// Initialize component without injecting PermIntlk interfaces
// This tests the scenario where PermIntlk configuration is not provided
TestComponent[5].Initialize();

// Since we never injected PermIntlk configuration interfaces,
// they should be null (0) by default
// The component should handle this gracefully via __QUERYINTERFACE checks

// Call CyclicLogic multiple times - should not crash
TestComponent[5].CyclicLogic();
TestComponent[5].CyclicLogic();

// Try to execute a command - should handle missing PermIntlk gracefully
TestComponent[5].ExecuteCommand(CmdIndex := 1);

// Component should still function
AssertTrue(
    Condition := TestComponent[5].BaseStatus.Initialized,
    Message := 'Component should remain initialized with missing PermIntlk interface'
);

// The command execution should not cause the component to crash
AssertFalse(
    Condition := TestComponent[5].BaseStatus.Error,
    Message := 'Component should not be in error state when PermIntlk interface is missing'
);

TEST_FINISHED();
END_METHOD

METHOD PRIVATE TEST_Component_QueryInterface_ValidatesTypes
VAR
    DummyCommandInterface : I_Command;
    QueryResult : BOOL;
END_VAR
// Tier 0 Test: Verify proper use of __QUERYINTERFACE for type checking
TEST(__POUNAME());

// Use array index 16 for this test method
iTestComponent := TestComponent[16];
iTestCommand := TestCommandConfigured[16].Command;

// Initialize test objects
TestComponent[16].Initialize();
TestCommandConfigured[16].Initialize();

// Test that the command implements I_Command interface
QueryResult := __QUERYINTERFACE(
    TestCommandConfigured[16].Command,
    DummyCommandInterface
);

AssertTrue(
    Condition := QueryResult,
    Message := 'FB_Command should implement I_Command interface'
);

// Test the pattern used in the codebase: check both != 0 AND __QUERYINTERFACE
// This is the defensive programming pattern used throughout the component
// Here we test with an actual interface reference, not a FB instance
AssertTrue(
    Condition := (TestCommandConfigured[16].iCommandConfiguration <> 0) AND __QUERYINTERFACE(TestCommandConfigured[16].iCommandConfiguration, TestCommandConfigured[16].iCommandConfiguration),
    Message := 'Standard pattern: interface should be non-null AND correct type'
);

// Verify that a null interface check properly fails
// The pattern (interface <> 0) protects against null access
AssertFalse(
    Condition := (0 <> 0),  // This is always FALSE when interface is null
    Message := 'Null check (0 <> 0) should be FALSE'
);

// This shows why we need the null check BEFORE __QUERYINTERFACE
// We don't call __QUERYINTERFACE on null to avoid potential issues

TEST_FINISHED();
END_METHOD

METHOD PRIVATE TEST_ComponentConfiguration_BaseConfiguration_ReferenceValid
// Tier 0 Test: ComponentConfiguration.BaseConfiguration reference should be valid
TEST(__POUNAME());

// Use array index 6 for this test method
iTestComponent := TestComponent[6];

// Initialize component
TestComponent[6].Initialize();

// Verify reference chain is valid
AssertTrue(
    Condition := __ISVALIDREF(TestComponent[6].ComponentConfiguration.BaseConfiguration),
    Message := 'ComponentConfiguration.BaseConfiguration reference should be valid'
);

// Verify the reference works by accessing a field through it
// Check that we can access nested fields without error
AssertTrue(
    Condition := TestComponent[6].ComponentConfiguration.BaseConfiguration.LogTraceConfiguration.When >= 0,
    Message := 'Should be able to access fields through BaseConfiguration reference'
);

TEST_FINISHED();
END_METHOD

METHOD PRIVATE TEST_ComponentStatus_BaseStatus_ReferenceValid
// Tier 0 Test: ComponentStatus.BaseStatus reference should be valid after init
TEST(__POUNAME());

// Use array index 7 for this test method
iTestComponent := TestComponent[7];

// Initialize component
TestComponent[7].Initialize();

// Verify reference chain is valid
AssertTrue(
    Condition := __ISVALIDREF(TestComponent[7].ComponentStatus.BaseStatus),
    Message := 'ComponentStatus.BaseStatus reference should be valid'
);

// Verify the reference is working by checking a value through it
AssertEquals_BOOL(
    Expected := TestComponent[7].BaseStatus.Initialized,
    Actual := TestComponent[7].ComponentStatus.BaseStatus.Initialized,
    Message := 'ComponentStatus.BaseStatus should reference component BaseStatus'
);

// Verify InitComplete is accessible through the reference
AssertTrue(
    Condition := TestComponent[7].ComponentStatus.BaseStatus.Initialized,
    Message := 'Should be able to access InitComplete through reference chain'
);

TEST_FINISHED();
END_METHOD

METHOD PRIVATE GivenAbortInvokedDuringValidation_CommandNeverEnqueuedOrExecuted
TEST(__POUNAME());

TEST_FINISHED();
END_METHOD

METHOD PRIVATE GivenBusyCommandElapsedTimeEqualsTimeout_CommandAborted
TEST(__POUNAME());

TEST_FINISHED();
END_METHOD

METHOD PRIVATE GivenCommandBusyAndInterlockLostWithAbortOnInterlockDrop_AbortFires
TEST(__POUNAME());

TEST_FINISHED();
END_METHOD

METHOD PRIVATE GivenCommandBusyAndInterlockLostWithoutAbortOnInterlockDrop_CommandContinues
TEST(__POUNAME());

TEST_FINISHED();
END_METHOD

METHOD PRIVATE GivenCommandBusyAndInterlockStaysOk_NoAbortOccurs
TEST(__POUNAME());

TEST_FINISHED();
END_METHOD

METHOD PRIVATE GivenComponentBusyDuringValidation_ResultConflict
TEST(__POUNAME());

TEST_FINISHED();
END_METHOD

METHOD PRIVATE GivenIndeterminantCommandDequeuedButPermissiveDropsBeforeExecute_ResultForbiddenNotOk
TEST(__POUNAME());

TEST_FINISHED();
END_METHOD

METHOD PRIVATE GivenInterlockNotInitComplete_CommandValidationFailsForbidden
TEST(__POUNAME());

TEST_FINISHED();
END_METHOD

METHOD PRIVATE GivenPermIntlkAllRequiredItemsTrue_EvaluateOKReturnsTrue
VAR
	// Test conditions that will all be TRUE
	TestCondition1							: BOOL := TRUE;
	TestCondition2							: BOOL := TRUE;
	TestCondition3							: BOOL := TRUE;
END_VAR
TEST(__POUNAME());

// Use array index 250 for this test method
iTestPermIntlkConfig := TestPermIntlkConfig[250];
iTestPermIntlk := TestPermIntlk[250];

// Configure PermIntlk for "All Conditions Must Be Met" mode
TestPermIntlkConfig[250].P_PermIntlkConfiguration.Mode := E_ModePermIntlk.IfAllConditionsMet;

// Set up multiple conditions that are all TRUE
TestPermIntlkConfig[250].P_PermIntlkConfiguration.PermIntlkObj[1].Condition := TestCondition1; // TRUE
TestPermIntlkConfig[250].P_PermIntlkConfiguration.PermIntlkObj[1].Description := 'Test Condition 1 - Should be TRUE';

TestPermIntlkConfig[250].P_PermIntlkConfiguration.PermIntlkObj[2].Condition := TestCondition2; // TRUE
TestPermIntlkConfig[250].P_PermIntlkConfiguration.PermIntlkObj[2].Description := 'Test Condition 2 - Should be TRUE';

TestPermIntlkConfig[250].P_PermIntlkConfiguration.PermIntlkObj[3].Condition := TestCondition3; // TRUE
TestPermIntlkConfig[250].P_PermIntlkConfiguration.PermIntlkObj[3].Description := 'Test Condition 3 - Should be TRUE';

// Initialize PermIntlk with configuration
TestPermIntlk[250].InjectPermIntlkConfiguration(iPermIntlkCfg := iTestPermIntlkConfig);
TestPermIntlk[250].Initialize();

// Verify initialization completed
AssertTrue(
    Condition := iTestPermIntlk.Initialized,
    Message := 'PermIntlk should be initialized after Initialize() called with valid config'
);

// Call Evaluate to process the conditions
iTestPermIntlk.Evaluate();

// Verify that P_OK returns TRUE when all required conditions are TRUE
AssertTrue(
    Condition := iTestPermIntlk.P_OK,
    Message := 'P_OK should return TRUE when all required conditions are TRUE in IfAllConditionsMet mode'
);

TEST_FINISHED();
END_METHOD

METHOD PRIVATE GivenPermIntlkInitNotComplete_EvaluateOKReturnsFalse
TEST(__POUNAME());

// Use array index 251 for this test method
iTestPermIntlk := TestPermIntlk[251];

// DO NOT call Initialize() on the PermIntlk - this simulates uninitialized state
// TestPermIntlk[251].Initialize(); // <-- Intentionally commented out

// Verify that InitComplete is FALSE (not initialized)
AssertFalse(
    Condition := iTestPermIntlk.Initialized,
    Message := 'PermIntlk should not be initialized when Initialize() not called'
);

// Call Evaluate to trigger evaluation logic
iTestPermIntlk.Evaluate();

// Verify that P_OK returns FALSE when not initialized
AssertFalse(
    Condition := iTestPermIntlk.P_OK,
    Message := 'P_OK should return FALSE when PermIntlk is not initialized'
);

TEST_FINISHED();
END_METHOD

METHOD PRIVATE GivenPermIntlkLostDuringBusy_WhenAbortOnInterlockDropFalse_CommandContinues
TEST(__POUNAME());

TEST_FINISHED();
END_METHOD

METHOD PRIVATE GivenPermIntlkOptionalItemFalse_EvaluateOKReturnsTrue
TEST(__POUNAME());

TEST_FINISHED();
END_METHOD

METHOD PRIVATE GivenPermIntlkRequiredItemFalse_EvaluateOKReturnsFalse
VAR	
	TestPermIntlkConfig						: FB_CmdPermIntlkConfiguration;
	iTestPermIntlkConfig					: I_PermIntlkConfiguration := TestPermIntlkConfig;
	
	TestPermIntlk							: FB_PermIntlk;
	iTestPermIntlk							: I_PermIntlk := TestPermIntlk;
	
	// Test conditions where one will be FALSE
	TestCondition1							: BOOL := TRUE;
	TestCondition2							: BOOL := FALSE; // This one FALSE should fail the entire check
	TestCondition3							: BOOL := TRUE;
END_VAR
TEST(__POUNAME());

// Configure PermIntlk for "All Conditions Must Be Met" mode
TestPermIntlkConfig.P_PermIntlkConfiguration.Mode := E_ModePermIntlk.IfAllConditionsMet;

// Set up conditions where one is FALSE
TestPermIntlkConfig.P_PermIntlkConfiguration.PermIntlkObj[1].Index := 1;
TestPermIntlkConfig.P_PermIntlkConfiguration.PermIntlkObj[1].Condition := TestCondition1; // TRUE
TestPermIntlkConfig.P_PermIntlkConfiguration.PermIntlkObj[1].Description := 'Test Condition 1 - Should be TRUE';

TestPermIntlkConfig.P_PermIntlkConfiguration.PermIntlkObj[2].Index := 2;
TestPermIntlkConfig.P_PermIntlkConfiguration.PermIntlkObj[2].Condition := TestCondition2; // FALSE - This should cause overall failure
TestPermIntlkConfig.P_PermIntlkConfiguration.PermIntlkObj[2].Description := 'Test Condition 2 - Should be FALSE (fails the test)';

TestPermIntlkConfig.P_PermIntlkConfiguration.PermIntlkObj[3].Index := 3;
TestPermIntlkConfig.P_PermIntlkConfiguration.PermIntlkObj[3].Condition := TestCondition3; // TRUE
TestPermIntlkConfig.P_PermIntlkConfiguration.PermIntlkObj[3].Description := 'Test Condition 3 - Should be TRUE';

// Initialize PermIntlk with configuration
TestPermIntlk.InjectPermIntlkConfiguration(iPermIntlkCfg := iTestPermIntlkConfig);
TestPermIntlk.Initialize();

// Verify initialization completed
AssertTrue(
    Condition := iTestPermIntlk.Initialized,
    Message := 'PermIntlk should be initialized after Initialize() called with valid config'
);

// Call Evaluate to process the conditions
iTestPermIntlk.Evaluate();

// Verify that P_OK returns FALSE when at least one required condition is FALSE
AssertFalse(
    Condition := iTestPermIntlk.P_OK,
    Message := 'P_OK should return FALSE when at least one required condition is FALSE in IfAllConditionsMet mode'
);

TEST_FINISHED();
END_METHOD

METHOD PRIVATE GivenPermissiveFalseDuringValidation_ResultForbidden
TEST(__POUNAME());

TEST_FINISHED();
END_METHOD

METHOD PRIVATE GivenResetCalledOnBusyCommand_ResultsInAbortThenNone
TEST(__POUNAME());

TEST_FINISHED();
END_METHOD

METHOD PRIVATE GivenAbortOnBusyCommand_LastCommandStatusUpdated
TEST(__POUNAME());

TEST_FINISHED();
END_METHOD

METHOD PRIVATE GivenAcceptedCommand_WhenExecuted_ResultBecomesOk
TEST(__POUNAME());

TEST_FINISHED();
END_METHOD

METHOD PRIVATE GivenBusyCommandElapsedTimeMeetsTimeout_WhenCmdTryCountEqualsConfiguredRetryCount_CommandIsAbortedAndMarkedTooManyRequests
TEST(__POUNAME());

TEST_FINISHED();
END_METHOD

METHOD PRIVATE GivenBusyCommandElapsedTimeMeetsTimeout_WhenCmdTryCountIsLessThanConfiguredRetryCount_CommandIsAbortedAndRequeued
TEST(__POUNAME());

TEST_FINISHED();
END_METHOD

METHOD PRIVATE GivenBusyCommandTimeoutBeforeRetry_RetryEnqueued
TEST(__POUNAME());

TEST_FINISHED();
END_METHOD

METHOD PRIVATE GivenBusyFlagTrueForAcceptedCommand_TurnsFalseOnlyAfterOkOrAbort
TEST(__POUNAME());

TEST_FINISHED();
END_METHOD

METHOD PRIVATE GivenCommandAborted_LastCommandStatusReflectsAbort
TEST(__POUNAME());

TEST_FINISHED();
END_METHOD

METHOD PRIVATE GivenCommandAborted_LastCommandStatusShowsAbortedUntilNextCommandRuns
TEST(__POUNAME());

TEST_FINISHED();
END_METHOD

METHOD PRIVATE GivenCommandAbortedThenReEnqueued_CommandTryCountResetsToPreviousPlusOne
TEST(__POUNAME());

TEST_FINISHED();
END_METHOD

METHOD PRIVATE GivenCommandAttemptsExceedRetryCount_ResultTooManyRequests
TEST(__POUNAME());

TEST_FINISHED();
END_METHOD

METHOD PRIVATE GivenCommandCompletes_CommandStatusDoneAndBusyCleared
TEST(__POUNAME());

TEST_FINISHED();
END_METHOD

METHOD PRIVATE GivenCommandExecutes_LastCommandStatusUpdatedToCurrentCommand
TEST(__POUNAME());

TEST_FINISHED();
END_METHOD

METHOD PRIVATE GivenCommandIsBusy_WhenNextCommandQueued_SecondCommandRemainsInQueue
TEST(__POUNAME());

TEST_FINISHED();
END_METHOD

METHOD PRIVATE GivenCommandPreempted_LastCommandStatusReflectsNewCommand
TEST(__POUNAME());

TEST_FINISHED();
END_METHOD

METHOD PRIVATE GivenCommandRetriesPastMaxAttempts_ResultTooManyRequests
TEST(__POUNAME());

TEST_FINISHED();
END_METHOD

METHOD PRIVATE GivenCommandTimesOutOnce_ResultRequestTimeout
TEST(__POUNAME());

TEST_FINISHED();
END_METHOD

METHOD PRIVATE GivenCreatedCommand_WhenDequeued_ResultIsAccepted
TEST(__POUNAME());

TEST_FINISHED();
END_METHOD

METHOD PRIVATE GivenEqualPriorityCommandQueued_ExistingBusyCommandNotAborted
TEST(__POUNAME());

TEST_FINISHED();
END_METHOD

METHOD PRIVATE GivenEqualPriorityCommandQueued_RunningCommandContinues
TEST(__POUNAME());

TEST_FINISHED();
END_METHOD

METHOD PRIVATE GivenExecutionTypeImmediateReturn_WhenDequeued_ResultTransitionsDirectlyToOkWithoutBusy
TEST(__POUNAME());

TEST_FINISHED();
END_METHOD

METHOD PRIVATE GivenExecutionTypeIndeterminant_WhenCommandValidated_ResultCreatedThenAcceptedThenBusy
TEST(__POUNAME());

TEST_FINISHED();
END_METHOD

METHOD PRIVATE GivenHigherPriorityCommandQueued_AbortsLowerPriorityRunningCommand
TEST(__POUNAME());

TEST_FINISHED();
END_METHOD

METHOD PRIVATE GivenIndeterminantCommandDequeued_ComponentBusyFlagSetTrueUntilCompletion
TEST(__POUNAME());

TEST_FINISHED();
END_METHOD

METHOD PRIVATE GivenNewCommandDequeued_LastCommandStatusSwitchesFromOldToNew
TEST(__POUNAME());

TEST_FINISHED();
END_METHOD

METHOD PRIVATE GivenNoBusyCommands_ComponentStatusBusyFalse
TEST(__POUNAME());

TEST_FINISHED();
END_METHOD

METHOD PRIVATE GivenOneBusyCommand_ComponentStatusBusyTrue
TEST(__POUNAME());

TEST_FINISHED();
END_METHOD

METHOD PRIVATE GivenQueuedCommand_ComponentStatusBusyFalseUntilExecution
TEST(__POUNAME());

TEST_FINISHED();
END_METHOD

METHOD PRIVATE GivenThatCommandIsBusyQueueNextCommand
TEST(__POUNAME());

TEST_FINISHED();
END_METHOD

METHOD PRIVATE GivenTimeoutZero_DisablesTimeoutLogic
TEST(__POUNAME());

TEST_FINISHED();
END_METHOD

METHOD PRIVATE GivenUseCommandPriorityFalse_NoPreemptionRegardlessOfPriority
TEST(__POUNAME());

TEST_FINISHED();
END_METHOD

METHOD PRIVATE GivenValidatedCommand_WhenEnqueued_ResultIsCreated
TEST(__POUNAME());

TEST_FINISHED();
END_METHOD

METHOD PRIVATE GivenAbortCalledTwice_IdempotentStateUnchangedSecondTime
TEST(__POUNAME());

TEST_FINISHED();
END_METHOD

METHOD PRIVATE GivenAllCommandInterfacesMissing_ComponentCyclicLogicDoesNotCrash
TEST(__POUNAME());

TEST_FINISHED();
END_METHOD

METHOD PRIVATE GivenChangingCommandConfigurationDuringBusyCommand_NoPointerCorruptionOrUnexpectedAbort
TEST(__POUNAME());

TEST_FINISHED();
END_METHOD

METHOD PRIVATE GivenCommandCancelledBeforeDequeued_ResultChangesToAbortedWithoutExecution
TEST(__POUNAME());

TEST_FINISHED();
END_METHOD

METHOD PRIVATE GivenCommandExecutesLongerThanConfiguredTimeoutButFinishes_SuccessfulCompletionOverridesTimeoutAbort
TEST(__POUNAME());

TEST_FINISHED();
END_METHOD

METHOD PRIVATE GivenCommandMarkedTooManyRequestsAndReset_AllowedToRequeueWithTryCountZero
TEST(__POUNAME());

TEST_FINISHED();
END_METHOD

METHOD PRIVATE GivenCommandResetWhileQueued_ResultChangesFromCreatedToNone
TEST(__POUNAME());

TEST_FINISHED();
END_METHOD

METHOD PRIVATE GivenComponentReset_AllChildReferencesRemainValid
TEST(__POUNAME());

TEST_FINISHED();
END_METHOD

METHOD PRIVATE GivenComponentReset_LastCommandStatusClearedOrResetAsConfigured
TEST(__POUNAME());

TEST_FINISHED();
END_METHOD

METHOD PRIVATE GivenComponentRestartWhileCommandsQueued_PendingQueueClearedOrRecoveredGracefully
TEST(__POUNAME());

TEST_FINISHED();
END_METHOD

METHOD PRIVATE GivenExceededRetryLimit_CommandResultTooManyRequestsAndNoRequeue
TEST(__POUNAME());

TEST_FINISHED();
END_METHOD

METHOD PRIVATE GivenInterlockNotConfigured_ValidationIgnoresPermIntlkPointer
TEST(__POUNAME());

TEST_FINISHED();
END_METHOD

METHOD PRIVATE GivenInvalidCmdIndex_ResultUnprocessableEntity
TEST(__POUNAME());

TEST_FINISHED();
END_METHOD

METHOD PRIVATE GivenInvalidCommand_ExpectError
VAR_INPUT
END_VAR
TEST(__POUNAME());

TEST_FINISHED();
END_METHOD

METHOD PRIVATE GivenInvalidCommandIndexGreaterThanUpperBound_ExecuteCommandReturnsUnprocessable
TEST(__POUNAME());

TEST_FINISHED();
END_METHOD

METHOD PRIVATE GivenLastCommandStatusUpdatedOnAbortThenOnNextExecute_NoStalePointer
TEST(__POUNAME());

TEST_FINISHED();
END_METHOD

METHOD PRIVATE GivenMissingCommandInterface_ResultUnprocessableEntity
TEST(__POUNAME());

TEST_FINISHED();
END_METHOD

METHOD PRIVATE GivenMissingConfigInterface_ResultUnprocessableEntity
TEST(__POUNAME());

TEST_FINISHED();
END_METHOD

METHOD PRIVATE GivenMissingPermIntlkInterface_ResultUnprocessableEntity
TEST(__POUNAME());

TEST_FINISHED();
END_METHOD

METHOD PRIVATE GivenNullComponentReferenceInCommand_ValidationAndExecutionNoOpsWithoutError
TEST(__POUNAME());

TEST_FINISHED();
END_METHOD

METHOD PRIVATE GivenNullPermIntlkPointer_WhenPermIntlkConfiguredFalse_ValidationPasses
TEST(__POUNAME());

TEST_FINISHED();
END_METHOD

METHOD PRIVATE GivenNullRingBufferPointer_WhenComponentExecutesValidation_NoNullPointerAccess
TEST(__POUNAME());

TEST_FINISHED();
END_METHOD

METHOD PRIVATE GivenPermIntlkNotLinkedToCommand_NoEvaluationOccursDuringCyclic
TEST(__POUNAME());

TEST_FINISHED();
END_METHOD

METHOD PRIVATE GivenPriorityOverflow_NoRuntimeException
TEST(__POUNAME());

TEST_FINISHED();
END_METHOD

METHOD PRIVATE GivenPriorityOverflowThenWrap_NoSchedulerCrash
TEST(__POUNAME());

TEST_FINISHED();
END_METHOD

METHOD PRIVATE GivenResetCalledOnCompletedCommand_StatusResetToNone
TEST(__POUNAME());

TEST_FINISHED();
END_METHOD

METHOD PRIVATE GivenRetryLimitExceededDuringValidation_ResultTooManyRequests
TEST(__POUNAME());

TEST_FINISHED();
END_METHOD

METHOD PRIVATE GivenRingBufferFull_WhenNewCommandEnqueued_ResultHeaderTooLarge
TEST(__POUNAME());

TEST_FINISHED();
END_METHOD

METHOD PRIVATE GivenRingBufferNotConfigured_EnqueueLogsFailure
TEST(__POUNAME());

TEST_FINISHED();
END_METHOD

METHOD PRIVATE GivenRingBufferWrapAround_NoCommandLostDuringContinuousEnqueueDequeue
TEST(__POUNAME());

TEST_FINISHED();
END_METHOD

METHOD PRIVATE GivenUnexpectedExceptionThrownInCommandExecute_ResultInternalServerErrorSetAndSystemContinues
TEST(__POUNAME());

TEST_FINISHED();
END_METHOD

METHOD PRIVATE GivenValidInterfaces_WhenComponentIdle_CommandValidatesContinues
TEST(__POUNAME());

TEST_FINISHED();
END_METHOD

METHOD PRIVATE GivenActiveCommand_CyclicLogicAlwaysCalledEachScan
TEST(__POUNAME());

TEST_FINISHED();
END_METHOD

METHOD PRIVATE GivenCommandAttemptedWithRetryCountEqualToConfiguredRetryCount_NoFurtherRetries
TEST(__POUNAME());

TEST_FINISHED();
END_METHOD

METHOD PRIVATE GivenCommandAttemptedWithRetryCountLessThanConfiguredRetryCount_RetryAllowed
TEST(__POUNAME());

TEST_FINISHED();
END_METHOD

METHOD PRIVATE GivenExecutionTypeImmediateReturn_WhenCommandValidated_ResultCreatedAndBusyNeverTrue
TEST(__POUNAME());

TEST_FINISHED();
END_METHOD

METHOD PRIVATE GivenExecutionTypeImmediateReturn_WhenTimeoutPeriodElapsed_NoTimeoutOccurs
TEST(__POUNAME());

TEST_FINISHED();
END_METHOD

METHOD PRIVATE GivenExecutionTypeIndeterminant_WhenBusyAndTimeoutExceeded_CommandRetriesOrFailsPerRetryCount
TEST(__POUNAME());

TEST_FINISHED();
END_METHOD

METHOD PRIVATE GivenHighPriorityCommandInsertedLate_PreemptsLowerPriorityBeforeExecutionStarts
TEST(__POUNAME());

TEST_FINISHED();
END_METHOD

METHOD PRIVATE GivenImmediateDequeueDisabled_CommandWaitsForNextCyclicExecution
TEST(__POUNAME());

TEST_FINISHED();
END_METHOD

METHOD PRIVATE GivenImmediateDequeueEnabled_CommandValidatedAndExecutedSameScan
TEST(__POUNAME());

TEST_FINISHED();
END_METHOD

METHOD PRIVATE GivenImmediateReturnAndIndeterminantInSameQueue_OrderOfCompletionReflectsQueueOrder
TEST(__POUNAME());

TEST_FINISHED();
END_METHOD

METHOD PRIVATE GivenImmediateReturnCommandDequeuedWhileComponentIdle_CompletesWithoutAffectingBusyFlag
TEST(__POUNAME());

TEST_FINISHED();
END_METHOD

METHOD PRIVATE GivenImmediateReturnCommandQueuedDuringBusyCommand_QueuesBehindButDoesNotPreempt
TEST(__POUNAME());

TEST_FINISHED();
END_METHOD

METHOD PRIVATE GivenImmediateReturnCommandQueuedWhileComponentBusy_CompletesInSameCycleAfterBusyClears
TEST(__POUNAME());

TEST_FINISHED();
END_METHOD

METHOD PRIVATE GivenImmediateReturnCommandWithAbortOnInterlockDropTrue_InterlockDropHasNoEffect
TEST(__POUNAME());

TEST_FINISHED();
END_METHOD

METHOD PRIVATE GivenImmediateReturnCommandWithZeroTimeout_DoesNotError
TEST(__POUNAME());

TEST_FINISHED();
END_METHOD

METHOD PRIVATE GivenInactiveCommand_CyclicLogicNotCalledToSaveCPU
TEST(__POUNAME());

TEST_FINISHED();
END_METHOD

METHOD PRIVATE GivenIndeterminantCommandWithZeroTimeout_TimesOutNextScan
TEST(__POUNAME());

TEST_FINISHED();
END_METHOD

METHOD PRIVATE GivenLowerPriorityCommandQueued_ReEnqueuedUntilRunningCommandFinishes
TEST(__POUNAME());

TEST_FINISHED();
END_METHOD

METHOD PRIVATE GivenMultipleCommandsHitTimeoutSimultaneously_AbortAndRetryOccursForEachCommandIndependently
TEST(__POUNAME());

TEST_FINISHED();
END_METHOD

METHOD PRIVATE GivenMultipleCommandsSamePriorityStartedSequentially_OnlyOneBusy
TEST(__POUNAME());

TEST_FINISHED();
END_METHOD

METHOD PRIVATE GivenMultipleImmediateReturnCommandsQueuedTogether_AllCompleteWithinSameScan
TEST(__POUNAME());

TEST_FINISHED();
END_METHOD

METHOD PRIVATE GivenMultipleLowerPriorityCommandsQueuedInBurst_ExecutionOrderPreservedFIFO
TEST(__POUNAME());

TEST_FINISHED();
END_METHOD

METHOD PRIVATE GivenNewHighPriorityCommandArrivesWhileBusy_OldCommandAbortedNewExecutes
TEST(__POUNAME());

TEST_FINISHED();
END_METHOD

METHOD PRIVATE GivenNoNewCommandsForNScans_LastCommandStatusRemainsUnchanged
TEST(__POUNAME());

TEST_FINISHED();
END_METHOD

METHOD PRIVATE GivenPermIntlkConfiguredAsFalse_CommandChecksOnlyAtStart_NoMidRunAbort
TEST(__POUNAME());

TEST_FINISHED();
END_METHOD

METHOD PRIVATE GivenPermIntlkConfiguredAsFalse_InterlockIgnoredDuringExecution
TEST(__POUNAME());

TEST_FINISHED();
END_METHOD

METHOD PRIVATE GivenPermIntlkEvaluateCalledEveryCycleWhileBusy_ToggleDetectedWithinOneScan
TEST(__POUNAME());

TEST_FINISHED();
END_METHOD

METHOD PRIVATE GivenPermIntlkFlappingRapidlyDuringBusyCommand_CommandAbortsOnlyAfterPersistentDrop
TEST(__POUNAME());

TEST_FINISHED();
END_METHOD

METHOD PRIVATE GivenPermIntlkFlapsLongerThanDebounce_AbortTriggered
TEST(__POUNAME());

TEST_FINISHED();
END_METHOD

METHOD PRIVATE GivenPermIntlkFlapsShorterThanDebounce_NoAbortTriggered
TEST(__POUNAME());

TEST_FINISHED();
END_METHOD

METHOD PRIVATE GivenPermIntlkTransitionFromFalseToTrue_EvaluateOKChangesAfterNextEvaluate
TEST(__POUNAME());

TEST_FINISHED();
END_METHOD

METHOD PRIVATE GivenPermissiveDropsForOneCycle_CommandNotAbortedUnlessDropPersists
TEST(__POUNAME());

TEST_FINISHED();
END_METHOD

METHOD PRIVATE GivenQueueContainsMixedPriorities_CorrectOrderRespectedEvenAfterReEnqueue
TEST(__POUNAME());

TEST_FINISHED();
END_METHOD

METHOD PRIVATE GivenReEnqueuedAfterTimeout_NewCommandResultIsCreated
TEST(__POUNAME());

TEST_FINISHED();
END_METHOD

METHOD PRIVATE GivenRetryCommandFinishesSuccessfully_PreviousTimeoutDoesNotBlockFutureEnqueue
TEST(__POUNAME());

TEST_FINISHED();
END_METHOD

METHOD PRIVATE GivenRetryTriggered_CommandReenqueuedAsNewQueueEntryWithIncrementedTryCount
TEST(__POUNAME());

TEST_FINISHED();
END_METHOD

METHOD PRIVATE GivenTimeoutAbort_LastCommandStatusReflectsRequestTimeoutReason
TEST(__POUNAME());

TEST_FINISHED();
END_METHOD

METHOD PRIVATE GivenTimeoutAfterFinalRetry_CommandStatusForeverTooManyRequestsUntilReset
TEST(__POUNAME());

TEST_FINISHED();
END_METHOD

METHOD PRIVATE GivenTimeoutAndRetryPolicyDisabled_CommandResetImmediately
TEST(__POUNAME());

TEST_FINISHED();
END_METHOD

METHOD PRIVATE GivenTimeoutRetryPath_ComponentBusyFlagClearsDuringAbortAndRemainsFalseUntilDequeuedAgain
TEST(__POUNAME());

TEST_FINISHED();
END_METHOD

METHOD PRIVATE GivenTimeoutValueShorterThanScanTime_CommandStillRetriesProperly
TEST(__POUNAME());

TEST_FINISHED();
END_METHOD

METHOD PRIVATE GivenTimeoutWithRetriesRemaining_CommandStatusFlipsAbortedThenCreatedWithinSameScan
TEST(__POUNAME());

TEST_FINISHED();
END_METHOD

END_FUNCTION_BLOCK

// Tests/FB_CommandConfigured/FB_CommandConfigured
{attribute 'no_explicit_call' := 'do not call this POU directly'}
FUNCTION_BLOCK FB_CommandConfigured EXTENDS FB_BaseCyclic
VAR
	Command					: FB_Command;
	CommandConfiguration 	: FB_CmdPermIntlkConfiguration;
	iCommandConfiguration	: I_CommandConfiguration := CommandConfiguration;
	iPermIntlkConfiguration	: I_PermIntlkConfiguration := CommandConfiguration;
END_VAR

END_FUNCTION_BLOCK

// Tests/MockFBs/FB_ComponentDerivative
{attribute 'no_explicit_call' := 'do not call this POU directly'}
FUNCTION_BLOCK FB_ComponentDerivative EXTENDS FB_Component<GC_Component.INDEX_COMMAND_MIN,GC_Component.INDEX_COMMAND_MAX>
VAR
END_VAR

PROPERTY P_TP_iSystemPermIntlk : REFERENCE TO I_PermIntlk
GET
P_TP_iSystemPermIntlk REF= _SystemPermIntlk;
END_GET
END_PROPERTY

METHOD PROTECTED _EvaluateCompletionConditions : BOOL
END_METHOD

(* Example implementation from FB_Actuator:
IF ActuatorStatus.ExtendOutput AND NOT ActuatorStatus.RetractOutput THEN
	ActuatorStatus.ActuatorState	:= E_ActuatorState.Extended;
ELSIF ActuatorStatus.RetractOutput AND NOT ActuatorStatus.ExtendOutput THEN
	ActuatorStatus.ActuatorState	:= E_ActuatorState.Retracted;
ELSE
	ActuatorStatus.ActuatorState	:= E_ActuatorState.Indeterminate;
END_IF

_UpdateComponentStatus := THIS^;*)
METHOD PROTECTED _UpdateComponentStatus : I_ComponentFull
END_METHOD

END_FUNCTION_BLOCK

// Tests/FB_CommandTestsII
FUNCTION_BLOCK FB_CommandTestsII EXTENDS TcUnit.FB_TestSuite
VAR CONSTANT
	// Test method index constants - one unique index per test method (0-113)

	// GivenCommand* helper test methods (0-25)
	INDEX_GIVENCOMMAND_WHENCANCEL_EXPECTREMOVEDFROMQUEUE							: DINT := 0;
	INDEX_GIVENCOMMAND_WHENCYCLICLOGICCALLED_EXPECTUPDATED							: DINT := 1;
	INDEX_GIVENCOMMAND_WHENEXECUTECALLED_EXPECTEXECUTION							: DINT := 2;
	INDEX_GIVENCOMMAND_WHENPAUSECALLED_EXPECTCOMMANDPAUSES							: DINT := 3;
	INDEX_GIVENCOMMAND_WHENQUEUECALLED_EXPECTADDEDTOQUEUE							: DINT := 4;
	INDEX_GIVENCOMMAND_WHENRESETCALLED_EXPECTSTATECLEARED							: DINT := 5;
	INDEX_GIVENCOMMAND_WHENRESUMECALLED_EXPECTCOMMANDRESUMES						: DINT := 6;
	INDEX_GIVENCOMMAND_WHENVALIDATECALLED_EXPECTPERMISSIVEOK						: DINT := 7;
	INDEX_GIVENCOMMAND_WHENVALIDATECALLED_EXPECTMATCHCONFIG							: DINT := 8;
	INDEX_GIVENCOMMANDALREADYRUNNING_WHENEXECUTE_CONFLICT							: DINT := 9;
	INDEX_GIVENCOMMANDEXECUTED_WHENCYCLICLOGICRUNS_EXPECTSTATEPROGRESSION			: DINT := 10;
	INDEX_GIVENCOMMANDINIDLESTATE_WHENCANCEL_EXPECTNOACTIONTAKEN					: DINT := 11;
	INDEX_GIVENCOMMANDINVALID_WHENVALIDATECALLED_EXPECTFALSE						: DINT := 12;
	INDEX_GIVENCOMMANDPAUSED_WHENABORT_EXPECTCOMMANDABORTEDANDSTATUSUPDATED			: DINT := 13;
	INDEX_GIVENCOMMANDPAUSED_WHENRESUME_EXPECTCOMMANDRESUMESEXECUTION				: DINT := 14;
	INDEX_GIVENCOMMANDQUEUED_WHENABORT_EXPECTCOMMANDABORTEDANDSTATUSUPDATED			: DINT := 15;
	INDEX_GIVENCOMMANDQUEUED_WHENCANCEL_EXPECTCOMMANDREMOVEDFROMQUEUE				: DINT := 16;
	INDEX_GIVENCOMMANDVALIDATED_WHENVALIDATECALLED_EXPECTTRUE						: DINT := 17;
	INDEX_GIVENCOMPONENTRESET_WHENRESETCALLED_EXPECTALLCOMMANDSTATECLEARED			: DINT := 18;
	INDEX_GIVENINJECTEDCONFIGURATIONSVALID_EXPECTINTERFACESSTOREDANDINITIALIZED		: DINT := 19;
	INDEX_GIVENINVALIDCONFIGURATION_WHENINJECTCONFIGURATIONCALLED_EXPECTINITFAILURE	: DINT := 20;
	INDEX_GIVENINVALIDCONFIGURATIONS_WHENINJECTCONFIGURATIONS_EXPECTINITFAILURE		: DINT := 21;
	INDEX_GIVENRUNNINGCOMMAND_WHENPAUSE_EXPECTCOMMANDTRANSITIONSTOPAUSEDSTATE		: DINT := 22;
	INDEX_GIVENTIMERSTARTED_WHENCYCLICLOGICRUNS_EXPECTELAPSEDTIMEINCREASES			: DINT := 23;
	INDEX_GIVENTIMERSTOPPED_WHENCYCLICLOGICRUNS_EXPECTELAPSEDTIMEREMAINCONSTANT		: DINT := 24;
	INDEX_GIVENVALIDCONFIGURATION_WHENINJECTCONFIGURATIONCALLED_EXPECTCONFIGSTORED	: DINT := 25;

	// TEST_* methods (26-113)
	INDEX_ABORT_AFTERCOMPLETE_IGNOREDWITHWARNING									: DINT := 26;
	INDEX_ABORT_ERRORCLASSIFICATION													: DINT := 27;
	INDEX_ABORT_WHENIDLEQUEUED_SETSRESULTABORTED									: DINT := 28;
	INDEX_ABORTAFTERCOMPLETE_STATEPRESERVATION										: DINT := 29;
	INDEX_ABORTDURINGCOMPLETIONWAIT													: DINT := 30;
	INDEX_ACCEPTEDCOMMAND_WHENEXECUTED_RESULTBECOMESOK								: DINT := 31;
	INDEX_BADREQUEST_INTERLOCKMISCONFIGURED											: DINT := 32;
	INDEX_BUSYCOMMANDELAPSEDTIMEEQUALS_COMMANDABORTED								: DINT := 33;
	INDEX_CANCEL_FROMQUEUEDSTATE													: DINT := 34;
	INDEX_CANCEL_REMOVESCOMMANDFROMQUEUE											: DINT := 35;
	INDEX_CANCEL_SETSCOMMANDSTATUSTOCANCELLED										: DINT := 36;
	INDEX_CANCEL_SETSRESULTCANCELLED												: DINT := 37;
	INDEX_CANCEL_WHENBUSY_REJECTED_NOCHANGETOSTATE									: DINT := 38;
	INDEX_COMMAND_LOCALREFERENCES_INITIALIZEDPROPERLY								: DINT := 39;
	INDEX_COMMAND_MISSINGCONFIGINTERFACE_FALLBACK									: DINT := 40;
	INDEX_COMMAND_PERMINTLKCHILD_INITIALIZED										: DINT := 41;
	INDEX_COMMANDATTEMPTSEXCEEDRETRYCOUNT											: DINT := 42;
	INDEX_COMMANDCOMPLETES_STATUSDONEANDCLEARED										: DINT := 43;
	INDEX_COMMANDSTATUS_CONFIGREF_POINTSTOCONFIGURATION								: DINT := 44;
	INDEX_COMMANDTIMEOUT_TRIGGERSRESET												: DINT := 45;
	INDEX_COMPLETE_ERROR_PERSISTSUNTILRESET											: DINT := 46;
	INDEX_COMPLETE_OK_AUTORESETNEXTCYCLE											: DINT := 47;
	INDEX_COMPLETESTATE_PRESERVESABORTEDRESULT										: DINT := 48;
	INDEX_COMPLETESTATE_PRESERVESTIMEOUTRESULT										: DINT := 49;
	INDEX_COMPLETESTATE_SETSOKFORSUCCESSFUL											: DINT := 50;
	INDEX_COMPLETIONCALLBACKTOSEQUENCER												: DINT := 51;
	INDEX_COMPLETIONCONDITIONEVALUATION												: DINT := 52;
	INDEX_COMPLETIONCONDITIONWITHTIMEOUT											: DINT := 53;
	INDEX_COMPLETIONWITHINTERLOCKDROP												: DINT := 54;
	INDEX_COMPLEXCOMPLETIONCONDITION												: DINT := 55;
	INDEX_COMPONENTBUSY_DURINGVALIDATION_RESULTCONFLICT								: DINT := 56;
	INDEX_CONFIG_FALLBACKTOLOCAL_WHENINJECTEDINVALID								: DINT := 57;
	INDEX_CONFIG_RECOVERYTOINJECTED_WHENVALIDAGAIN									: DINT := 58;
	INDEX_CONFIGURATIONRESOLUTION_HANDLESVALIDINVALID								: DINT := 59;
	INDEX_CYCLICLOGIC_STATEMACHINEPROGRESSION										: DINT := 60;
	INDEX_DISCRETECOMPLETIONCONDITION												: DINT := 61;
	INDEX_DYNAMICCOMPLETIONCONDITIONUPDATE											: DINT := 62;
	INDEX_EDGETRIGGERED_STATEMACHINEEXECUTION										: DINT := 63;
	INDEX_EXECUTE_HAPPYPATH_TRANSITIONSTOMONITOR									: DINT := 64;
	INDEX_EXECUTE_STATEMACHINEPROGRESSION											: DINT := 65;
	INDEX_EXECUTE_TRANSITIONSFROMACCEPTEDTOOK										: DINT := 66;
	INDEX_EXECUTE_VALIDATESBEFOREACCEPTING											: DINT := 67;
	INDEX_EXECUTE_WHENPERMISSIVEMISSING_RETURNSFORBIDDEN							: DINT := 68;
	INDEX_FASTCOMPLETIONINONESCAN													: DINT := 69;
	INDEX_FORBIDDEN_RESUMEWITHOUTPERMISSIVE											: DINT := 70;
	INDEX_INJECTCONFIGURATIONS_STORESINTERFACES										: DINT := 71;
	INDEX_INTERFACEINJECTIONCONFIGURATIONRESOLUTION									: DINT := 72;
	INDEX_INTERLOCKDROP_ABORTSCOMMANDWHENCONFIGURED									: DINT := 73;
	INDEX_INTERLOCKDROP_FROMMONITORSTATE											: DINT := 74;
	INDEX_INTERLOCKINVALIDCONFIG_DURINGVALIDATION									: DINT := 75;
	INDEX_INTERLOCKLOST_COMPREHENSIVESTATETRANSITIONS								: DINT := 76;
	INDEX_INTERLOCKLOST_FROMEXECUTESTATE											: DINT := 77;
	INDEX_INTERLOCKLOST_SETSCORRECTRESULT											: DINT := 78;
	INDEX_INTERLOCKREFERENCELOST_DURINGEXECUTION									: DINT := 79;
	INDEX_METHODENABLEMENT_BUSYSTATE_ALLOWABORT										: DINT := 80;
	INDEX_METHODENABLEMENT_DONESTATE_ALLOWRESET										: DINT := 81;
	INDEX_METHODENABLEMENT_IDLEWITHINTERLOK_ALLOWEXECUTE							: DINT := 82;
	INDEX_METHODENABLEMENT_IDLEWITHOUTINTERLOK_REJECT								: DINT := 83;
	INDEX_MOTIONCOMPLETIONCONDITION													: DINT := 84;
	INDEX_OPERATIONTOCOMMANDTRANSLATION												: DINT := 85;
	INDEX_OPERATORABORT_VSINTERLOCKABORT_DIFFERENTRESULTS							: DINT := 86;
	INDEX_PAUSERESUME_STATETRANSITIONS												: DINT := 87;
	INDEX_PAUSERESUMEWITHCOMPLETIONCONDITION										: DINT := 88;
	INDEX_PERMINTLKLOST_DURINGBUSY_COMMANDABORTED									: DINT := 89;
	INDEX_PERMISSIVEFALSE_DURINGVALIDATION_FORBIDDEN								: DINT := 90;
	INDEX_QUEUEOPERATIONS_MULTIPLECOMMANDSATOMICITY									: DINT := 91;
	INDEX_RECIPEMANAGERPROVIDESCOMMANDCONFIG										: DINT := 92;
	INDEX_RESET_CLEARSCOMMANDSTATE													: DINT := 93;
	INDEX_RESULTPERSISTENCE_TERMINALSTATES											: DINT := 94;
	INDEX_RETRYCOUNT_INCREMENTONEXECUTIONSTARTONLY									: DINT := 95;
	INDEX_RUNTIMECOMMANDCONFIGLOSS_INJECTEDREFSINVALIDATED							: DINT := 96;
	INDEX_RUNTIMECOMMANDCONFIGRECOVERY_VALIDREFSRESTORED							: DINT := 97;
	INDEX_SLOWCOMPLETIONMULTIPLESCANS												: DINT := 98;
	INDEX_STEPSTATE_TRANSITIONSANDVALIDATION										: DINT := 99;
	INDEX_SYSTEMATICSTATEVALIDATION_IDLESTATES										: DINT := 100;
	INDEX_SYSTEMATICSTATEVALIDATION_TERMINALSTATES									: DINT := 101;
	INDEX_TERMINALRESULTS_ERRORFLAGCONSISTENCY										: DINT := 102;
	INDEX_TIMEBASEDCOMPLETIONCONDITION												: DINT := 103;
	INDEX_TIMEOUTANDINTERLOCKLOST_SAMECYCLE_PRIORITIZE								: DINT := 104;
	INDEX_TIMERCOMPLETIONTIME_SETONCOMMANDCOMPLETE									: DINT := 105;
	INDEX_TIMERINTEGRATION_WITHCOMMANDSTATEMACHINE									: DINT := 106;
	INDEX_TIMERPAUSERESUME_ELAPSEDTIMEACCURACY										: DINT := 107;
	INDEX_TIMERSTOPSONCOMMANDCOMPLETE_NOTTIMEOUT									: DINT := 108;
	INDEX_TIMERTRIGGERTIME_SETONCOMMANDSTART										: DINT := 109;
	INDEX_VALIDATE_RETURNSPROPERRESULT												: DINT := 110;
	INDEX_VALIDATE_WITHCONTINUOUSEVALUATION											: DINT := 111;
	INDEX_VALIDATIONOK_INTERLOCKDROP_DURINGEXECUTION								: DINT := 112;
	INDEX_VALIDCOMMAND_EXPECTEXECUTED												: DINT := 113;

	// Additional indices for multi-scenario tests
	INDEX_TERMINALRESULTS_CLEANCANCEL												: DINT := 114;
	INDEX_TERMINALRESULTS_INTERLOCKLOST											: DINT := 115;
	INDEX_TERMINALRESULTS_TIMEOUT													: DINT := 116;
	INDEX_TERMINALRESULTS_COMPLETE_OK												: DINT := 117;
	INDEX_TERMINALRESULTS_COMPLETE_ERROR											: DINT := 118;
	INDEX_VALIDATIONOK_INTERLOCKDROP_SCENARIO2										: DINT := 119;

	// Fixed duplicate indices - these tests were incorrectly reusing other test indices
	INDEX_TIMEOUTANDINTERLOCKLOST_SAMECYCLE_PRIORITIZEINTERLOCKLOST					: DINT := 120;
	INDEX_VALIDATE_RETURNSPROPERRESULTBASEDONPERMISSIVES							: DINT := 121;
	INDEX_VALIDATE_WITHCONTINUOUSEVALUATION_PROPER									: DINT := 122;
	INDEX_VALIDATIONOK_INTERLOCKDROPDURINGEXECUTION									: DINT := 123;
	INDEX_VALIDCOMMAND_EXPECTEXECUTED_PROPER										: DINT := 124;
END_VAR

VAR

	// Mock component for testing
	MockComponent 			: FB_ComponentDerivative;

	// Common test interfaces for all methods (FB-level for stability)
	// Initialized to 0 to prevent page faults - will be set by each test method safely
	iTestCommand 			: I_CommandUnderTest;
	iTestCommandConfig 		: I_CommandConfiguration;
	iTestComponent 			: I_ComponentFull;
	iTestPermIntlkConfig 	: I_PermIntlkConfiguration;
	iTestPermIntlk 			: I_PermIntlk;
	iTestPermIntlkEval		: I_PermIntlk;
	
	// Array instances for test methods (indices 0-17)
	TestCommand : ARRAY[GC_Test.INDEX_TestFB_Command_MIN..GC_Test.INDEX_TestFB_Command_MAX] OF FB_CommandUnderTest;
	TestComponent : ARRAY[GC_Test.INDEX_TestFB_Command_MIN..GC_Test.INDEX_TestFB_Command_MAX] OF FB_ComponentDerivative;
	TestCommandConfig : ARRAY[GC_Test.INDEX_TestFB_Command_MIN..GC_Test.INDEX_TestFB_Command_MAX] OF FB_CmdPermIntlkConfiguration;
	TestPermIntlk : ARRAY[GC_Test.INDEX_TestFB_Command_MIN..GC_Test.INDEX_TestFB_Command_MAX] OF FB_PermIntlkCommand;
	MockQueue : ARRAY[GC_Test.INDEX_TestFB_Command_MIN..GC_Test.INDEX_TestFB_Command_MAX] OF FB_RingBufferICmd;
	CommandTimer : ARRAY[GC_Test.INDEX_TestFB_Command_MIN..GC_Test.INDEX_TestFB_Command_MAX] OF FB_CommandElapsedTimer;
//	FileHandler : ARRAY[GC_Test.INDEX_TestFB_Command_MIN..GC_Test.INDEX_TestFB_Command_MAX] OF FB_FileHandlerCsv;
END_VAR

// ================================================================
// ACTIVE TESTS - BehaviorTests, FaultInjectionTests, StateDrivenCompletenessTests, IntegrationTests
// ================================================================

// Tests before systematic state coverage section are in FB_CommandTestsI

// SYSTEMATIC STATE COVERAGE TESTS - New systematic approach for 128 truth table combinations
TEST_SystematicStateValidation_IdleStates();
TEST_SystematicStateValidation_TerminalStates();
//TEST_QueueOperations_MultipleCommandsAtomicity();
TEST_Execute_ValidatesBeforeAccepting();
TEST_Complete_Ok_AutoResetsNextCycle();
TEST_Complete_Error_PersistsUntilReset();
TEST_Cancel_WhenBusy_RejectedWithWarning_NoStateChange();

TEST_RetryCount_IncrementOnExecutionStartOnly();
TEST_Config_FallbackToLocal_WhenInjectedInvalid();
TEST_Config_RecoveryToInjected_WhenValidAgain();

// === Unified Command Completion Condition Tests ===
TEST_FastCompletionInOneScan();

TEST_CompletionConditionEvaluation();
TEST_RecipeManagerProvidesCommandConfig();
TEST_OperationToCommandTranslation();
TEST_MotionCompletionCondition();
TEST_DiscreteCompletionCondition();
TEST_TimeBasedCompletionCondition();
TEST_CompletionWithInterlockDrop();

TEST_CompletionCallbackToSequencer();
TEST_AbortDuringCompletionWait();

TEST_DynamicCompletionConditionUpdate();

// Runtime configuration loss tests - validate actual fix scenarios
TEST_RuntimeCommandConfigLoss_InjectedRefsInvalidatedDuringExecution();
TEST_RuntimeCommandConfigRecovery_ValidRefsRestoredDuringExecution();
TEST_TimeoutAndInterlockLost_SameCycle_PrioritizeInterlockLost();
TEST_Abort_AfterComplete_IgnoredWithWarning();
TEST_Abort_WhenIdleQueued_SetsResultAbortedAndRemovesFromQueue();
TEST_Execute_HappyPath_TransitionsToMonitorAndCompletesOk();
TEST_Execute_WhenPermissiveMissing_ReturnsForbidden();

METHOD PRIVATE TEST_Abort_AfterComplete_IgnoredWithWarning
VAR
	TestIdx : DINT := INDEX_ABORT_AFTERCOMPLETE_IGNOREDWITHWARNING;
	CompletionCondition	: BOOL;
END_VAR
VAR_INPUT
END_VAR
TEST(__POUNAME());

// This test verifies that calling Abort() after a command has already completed should be ignored
// The command should remain in Complete state with Ok result (terminal state protection)

// Initialize test objects
TestCommand[TestIdx].Initialize();
TestComponent[TestIdx].Initialize();
TestCommandConfig[TestIdx].Initialize();
TestPermIntlk[TestIdx].Initialize();

// Safe interface assignments
iTestCommand := TestCommand[TestIdx];
iTestCommandConfig := TestCommandConfig[TestIdx];
iTestComponent := TestComponent[TestIdx];
iTestPermIntlkConfig := TestPermIntlk[TestIdx];

// Interface validation with protection
IF iTestCommand = 0 THEN
	AssertTrue(Condition := FALSE, Message := 'TEST FAILED: iTestCommand interface is null');
	RETURN;
END_IF

IF iTestCommandConfig = 0 THEN
	AssertTrue(Condition := FALSE, Message := 'TEST FAILED: iTestCommandConfig interface is null');
	RETURN;
END_IF

IF iTestComponent = 0 THEN
	AssertTrue(Condition := FALSE, Message := 'TEST FAILED: iTestComponent interface is null');
	RETURN;
END_IF

// Configure command with immediate completion
CompletionCondition	:= TRUE;
iTestCommandConfig.P_CommandConfiguration.CompletionCondition REF= CompletionCondition;
iTestCommandConfig.P_CommandConfiguration.CommandDescription := 'Abort after complete test';
iTestCommandConfig.P_CommandConfiguration.TimeoutTime := T#30S;
IF __ISVALIDREF(iTestCommandConfig.P_CommandConfiguration.BaseConfiguration) THEN
	iTestCommandConfig.P_CommandConfiguration.BaseConfiguration.LogTraceConfiguration.When := E_LogTraceWhen.xRunOnInitOnly;
END_IF

// Setup component to be enabled and not busy
IF iTestComponent <> 0 THEN
	iTestComponent.P_ComponentStatus.BaseStatus.Enabled := TRUE;
	iTestComponent.P_ComponentStatus.BaseStatus.Busy := FALSE;
	iTestComponent.P_ComponentStatus.BaseStatus.Error := FALSE;
END_IF

// Configure permissive to be OK
IF iTestPermIntlkConfig <> 0 THEN
	iTestPermIntlkConfig.P_PermIntlkConfiguration.PermIntlkObj[1].Description := 'Abort After Complete Permissive';
	iTestPermIntlkConfig.P_PermIntlkConfiguration.PermIntlkObj[1].Condition := TRUE;
	iTestPermIntlkConfig.P_PermIntlkConfiguration.PermIntlkObj[1].Index := 1;
	TestPermIntlk[TestIdx].CyclicLogic(); // Update permissive evaluation
END_IF

// Setup command with configurations
iTestCommand.InjectConfigurations(
	iComponent := iTestComponent,
	iCommandConfiguration := iTestCommandConfig,
	iPermIntlkConfiguration := iTestPermIntlkConfig
);

// Resolve configurations after injection
iTestCommand.CyclicLogic();

// Execute command
iTestCommand.Execute();

// Progress through state machine to completion
iTestCommand.CyclicLogic(); // Idle → Execute
iTestCommand.CyclicLogic(); // Execute → Monitor
iTestCommand.Complete(); // Signal completion
iTestCommand.CyclicLogic(); // Monitor → Complete

// Verify command completed successfully
AssertEquals_UDINT(
	Expected := E_CommandState.Complete,
	Actual := iTestCommand.P_CommandStatus.StepState,
	Message := 'Command should be in Complete state before attempting Abort'
);

AssertEquals_UDINT(
	Expected := E_CommandResult.Ok,
	Actual := iTestCommand.P_CommandStatus.Result,
	Message := 'Command should have Result=Ok after successful completion'
);

AssertTrue(
	Condition := iTestCommand.P_CommandStatus.BaseStatus.Done,
	Message := 'Command should have Done=TRUE after completion'
);

// Now attempt to abort the already-completed command
iTestCommand.Abort();

// Verify that Abort() is ignored - command remains in Complete state with Ok result
AssertEquals_UDINT(
	Expected := E_CommandState.Complete,
	Actual := iTestCommand.P_CommandStatus.StepState,
	Message := 'TERMINAL STATE PROTECTION: Command should remain in Complete state after Abort attempt'
);

AssertEquals_UDINT(
	Expected := E_CommandResult.Ok,
	Actual := iTestCommand.P_CommandStatus.Result,
	Message := 'TERMINAL STATE PROTECTION: Result should remain Ok (not overwritten to Aborted)'
);

AssertTrue(
	Condition := iTestCommand.P_CommandStatus.BaseStatus.Done,
	Message := 'Done flag should remain TRUE after ignored Abort attempt'
);

TEST_FINISHED();
END_METHOD

METHOD PRIVATE TEST_Abort_WhenIdleQueued_SetsResultAbortedAndRemovesFromQueue
VAR
	TestIdx : DINT := INDEX_ABORT_WHENIDLEQUEUED_SETSRESULTABORTED;
	CompletionCondition	: BOOL;
END_VAR
TEST(__POUNAME());

// This test verifies that calling Abort() on a command in Idle or Queued state
// properly sets Result=Aborted and cleans up any queue state

// Initialize test objects
TestCommand[TestIdx].Initialize();
TestComponent[TestIdx].Initialize();
TestCommandConfig[TestIdx].Initialize();
TestPermIntlk[TestIdx].Initialize();

// Safe interface assignments
iTestCommand := TestCommand[TestIdx];
iTestCommandConfig := TestCommandConfig[TestIdx];
iTestComponent := TestComponent[TestIdx];
iTestPermIntlkConfig := TestPermIntlk[TestIdx];

// Interface validation with protection
IF iTestCommand = 0 THEN
	AssertTrue(Condition := FALSE, Message := 'TEST FAILED: iTestCommand interface is null');
	RETURN;
END_IF

IF iTestCommandConfig = 0 THEN
	AssertTrue(Condition := FALSE, Message := 'TEST FAILED: iTestCommandConfig interface is null');
	RETURN;
END_IF

IF iTestComponent = 0 THEN
	AssertTrue(Condition := FALSE, Message := 'TEST FAILED: iTestComponent interface is null');
	RETURN;
END_IF

// Configure command
CompletionCondition	:= FALSE;
iTestCommandConfig.P_CommandConfiguration.CompletionCondition REF= CompletionCondition;
iTestCommandConfig.P_CommandConfiguration.CommandDescription := 'Abort when Idle/Queued test';
iTestCommandConfig.P_CommandConfiguration.TimeoutTime := T#30S;
IF __ISVALIDREF(iTestCommandConfig.P_CommandConfiguration.BaseConfiguration) THEN
	iTestCommandConfig.P_CommandConfiguration.BaseConfiguration.LogTraceConfiguration.When := E_LogTraceWhen.xRunOnInitOnly;
END_IF

// Setup component to be enabled and not busy
IF iTestComponent <> 0 THEN
	iTestComponent.P_ComponentStatus.BaseStatus.Enabled := TRUE;
	iTestComponent.P_ComponentStatus.BaseStatus.Busy := FALSE;
	iTestComponent.P_ComponentStatus.BaseStatus.Error := FALSE;
END_IF

// Configure permissive to be OK
IF iTestPermIntlkConfig <> 0 THEN
	iTestPermIntlkConfig.P_PermIntlkConfiguration.PermIntlkObj[1].Description := 'Abort Idle/Queued Permissive';
	iTestPermIntlkConfig.P_PermIntlkConfiguration.PermIntlkObj[1].Condition := TRUE;
	iTestPermIntlkConfig.P_PermIntlkConfiguration.PermIntlkObj[1].Index := 1;
	TestPermIntlk[TestIdx].CyclicLogic(); // Update permissive evaluation
END_IF

// Setup command with configurations
iTestCommand.InjectConfigurations(
	iComponent := iTestComponent,
	iCommandConfiguration := iTestCommandConfig,
	iPermIntlkConfiguration := iTestPermIntlkConfig
);

// Resolve configurations after injection
iTestCommand.CyclicLogic();

// === TEST CASE 1: Abort command while in Idle state (before Execute) ===
// Verify starting in Idle state
AssertEquals_UDINT(
	Expected := E_CommandState.Idle,
	Actual := iTestCommand.P_CommandStatus.StepState,
	Message := 'Command should start in Idle state'
);

// Attempt to abort while in Idle state
iTestCommand.Abort();

// Verify Abort sets Result=Aborted even from Idle state
AssertEquals_UDINT(
	Expected := E_CommandResult.Aborted,
	Actual := iTestCommand.P_CommandStatus.Result,
	Message := 'Abort from Idle state should set Result=Aborted'
);

AssertEquals_UDINT(
	Expected := E_CommandState.Idle,
	Actual := iTestCommand.P_CommandStatus.StepState,
	Message := 'Command should remain in Idle state after Abort from Idle'
);

// === TEST CASE 2: Queue command and then abort ===
// Reset command for next test
iTestCommand.Reset();

// Queue the command (if Queue method exists, otherwise simulate)
iTestCommand.Queue();

// Verify command is queued or in Idle state (depending on implementation)
// The test name suggests command should be removed from queue

// Abort the queued command
iTestCommand.Abort();

// Verify Abort properly cleans up queued state
AssertEquals_UDINT(
	Expected := E_CommandResult.Aborted,
	Actual := iTestCommand.P_CommandStatus.Result,
	Message := 'Abort should set Result=Aborted for queued command'
);

AssertFalse(
	Condition := iTestCommand.P_CommandStatus.BaseStatus.Busy,
	Message := 'Aborted queued command should not be Busy'
);

// Verify command is removed from queue (no longer pending execution)
AssertEquals_UDINT(
	Expected := E_CommandState.Idle,
	Actual := iTestCommand.P_CommandStatus.StepState,
	Message := 'Aborted command should be in Idle state (removed from queue)'
);

TEST_FINISHED();
END_METHOD

METHOD PRIVATE TEST_Cancel_WhenBusy_RejectedWithWarning_NoStateChange
VAR
	TestIdx : DINT := INDEX_CANCEL_WHENBUSY_REJECTED_NOCHANGETOSTATE;
    initialResult : E_CommandResult;
    initialState : E_CommandState;
    initialBusy : BOOL;
    initialDone : BOOL;
    initialError : BOOL;
END_VAR
TEST(__POUNAME());

// Purpose: Verify Cancel is properly rejected when command is busy
// Tests guard condition: Cancel only allowed when NOT Busy AND NOT Error AND NOT Done

// Initialize test objects - Use index 20
TestCommand[TestIdx].Initialize();
TestComponent[TestIdx].Initialize();
TestCommandConfig[TestIdx].Initialize();
TestPermIntlk[TestIdx].Initialize();

// Safe interface assignments - check for non-null
iTestCommand := TestCommand[TestIdx];

iTestCommandConfig := TestCommandConfig[TestIdx];

iTestComponent := TestComponent[TestIdx];

iTestPermIntlkConfig := TestPermIntlk[TestIdx];

// Interface validation
IF iTestCommand = 0 THEN
    AssertTrue(Condition := FALSE, Message := 'TEST FAILED: iTestCommand interface is null');
    RETURN;
END_IF

// Configure command
TestCommandConfig[TestIdx].P_CommandConfiguration.CommandDescription := 'Cancel Busy Test';
TestCommandConfig[TestIdx].P_CommandConfiguration.TimeoutTime := T#30S;
IF __ISVALIDREF(TestCommandConfig[TestIdx].P_CommandConfiguration.BaseConfiguration) THEN
    TestCommandConfig[TestIdx].P_CommandConfiguration.BaseConfiguration.LogTraceConfiguration.When := E_LogTraceWhen.xRunOnInitOnly;
END_IF

// Configure permissive to be OK for successful validation and execution
IF iTestPermIntlkConfig <> 0 THEN
	iTestPermIntlkConfig.P_PermIntlkConfiguration.PermIntlkObj[1].Description := 'Cancel Test Permissive';
	iTestPermIntlkConfig.P_PermIntlkConfiguration.PermIntlkObj[1].Condition := TRUE;
	iTestPermIntlkConfig.P_PermIntlkConfiguration.PermIntlkObj[1].Index := 1;
	TestPermIntlk[TestIdx].CyclicLogic(); // Update permissive evaluation
END_IF

// Setup command with configurations
iTestCommand.InjectConfigurations(
    iComponent := iTestComponent,
    iCommandConfiguration := iTestCommandConfig,
    iPermIntlkConfiguration := iTestPermIntlkConfig
);

// Resolve configurations after injection
iTestCommand.CyclicLogic();

// === STEP 1: Make Command Busy ===
iTestCommand.Execute();
iTestCommand.CyclicLogic(); // Transition to Execute state

// Verify command is busy
AssertTrue(
    Condition := iTestCommand.P_CommandStatus.BaseStatus.Busy,
    Message := 'Command should be busy before testing Cancel rejection'
);

AssertEquals_UDINT(
    Expected := E_CommandState.Execute,
    Actual := iTestCommand.P_CommandStatus.StepState,
    Message := 'Command should be in Execute state'
);

// === STEP 2: Capture Initial State Before Cancel Attempt ===
initialResult := iTestCommand.P_CommandStatus.Result;
initialState := iTestCommand.P_CommandStatus.StepState;
initialBusy := iTestCommand.P_CommandStatus.BaseStatus.Busy;
initialDone := iTestCommand.P_CommandStatus.BaseStatus.Done;
initialError := iTestCommand.P_CommandStatus.BaseStatus.Error;

// === STEP 3: Attempt Cancel While Busy ===
iTestCommand.Cancel();

// === STEP 4: Verify Cancel Was Rejected and State Unchanged ===
AssertEquals_UDINT(
    Expected := initialResult,
    Actual := iTestCommand.P_CommandStatus.Result,
    Message := 'POLICY: Cancel should not change Result when command is busy'
);

AssertEquals_UDINT(
    Expected := initialState,
    Actual := iTestCommand.P_CommandStatus.StepState,
    Message := 'POLICY: Cancel should not change State when command is busy'
);

AssertEquals_BOOL(
    Expected := initialBusy,
    Actual := iTestCommand.P_CommandStatus.BaseStatus.Busy,
    Message := 'POLICY: Cancel should not change Busy flag when command is busy'
);

AssertEquals_BOOL(
    Expected := initialDone,
    Actual := iTestCommand.P_CommandStatus.BaseStatus.Done,
    Message := 'POLICY: Cancel should not change Done flag when command is busy'
);

AssertEquals_BOOL(
    Expected := initialError,
    Actual := iTestCommand.P_CommandStatus.BaseStatus.Error,
    Message := 'POLICY: Cancel should not change Error flag when command is busy'
);

// === STEP 5: Command Should Continue Normal Execution ===
iTestCommand.CyclicLogic(); // Execute → Monitor
AssertEquals_UDINT(
    Expected := E_CommandState.Monitor,
    Actual := iTestCommand.P_CommandStatus.StepState,
    Message := 'Command should continue normal execution after rejected Cancel'
);

iTestCommand.Complete(); // Signal completion
iTestCommand.CyclicLogic(); // Monitor → Complete
AssertEquals_UDINT(
    Expected := E_CommandState.Complete,
    Actual := iTestCommand.P_CommandStatus.StepState,
    Message := 'Command should complete normally after rejected Cancel'
);

AssertEquals_UDINT(
    Expected := E_CommandResult.Ok,
    Actual := iTestCommand.P_CommandStatus.Result,
    Message := 'Command should complete with Ok result after rejected Cancel'
);

// === STEP 6: Test Cancel Works When Command is Idle ===
// Auto-reset requires 2 cycles in Complete state
iTestCommand.CyclicLogic(); // First cycle in Complete (stays Complete)
iTestCommand.CyclicLogic(); // Second cycle in Complete (auto-resets to Idle)

// Verify command is now idle and not busy
AssertEquals_UDINT(
    Expected := E_CommandState.Idle,
    Actual := iTestCommand.P_CommandStatus.StepState,
    Message := 'Command should be Idle for positive cancel test'
);

AssertFalse(
    Condition := iTestCommand.P_CommandStatus.BaseStatus.Busy,
    Message := 'Command should not be busy for positive cancel test'
);

// Cancel should work when not busy
iTestCommand.Cancel();

AssertEquals_UDINT(
    Expected := E_CommandResult.Cancelled,
    Actual := iTestCommand.P_CommandStatus.Result,
    Message := 'POSITIVE TEST: Cancel should work when command is not busy'
);

TEST_FINISHED();
END_METHOD

METHOD PRIVATE TEST_Execute_HappyPath_TransitionsToMonitorAndCompletesOk : REFERENCE TO FB_Test
VAR
	TestIdx : DINT := INDEX_EXECUTE_HAPPYPATH_TRANSITIONSTOMONITOR;
	CompletionCondition	: BOOL;
END_VAR
VAR_INPUT
END_VAR
TEST(__POUNAME());

// This test verifies the happy path execution flow:
// Idle → Execute → Monitor → Complete with Result=Ok

// Initialize test objects
TestCommand[TestIdx].Initialize();
TestComponent[TestIdx].Initialize();
TestCommandConfig[TestIdx].Initialize();
TestPermIntlk[TestIdx].Initialize();

// Safe interface assignments
iTestCommand := TestCommand[TestIdx];
iTestCommandConfig := TestCommandConfig[TestIdx];
iTestComponent := TestComponent[TestIdx];
iTestPermIntlkConfig := TestPermIntlk[TestIdx];

// Interface validation with protection
IF iTestCommand = 0 THEN
	AssertTrue(Condition := FALSE, Message := 'TEST FAILED: iTestCommand interface is null');
	RETURN;
END_IF

IF iTestCommandConfig = 0 THEN
	AssertTrue(Condition := FALSE, Message := 'TEST FAILED: iTestCommandConfig interface is null');
	RETURN;
END_IF

IF iTestComponent = 0 THEN
	AssertTrue(Condition := FALSE, Message := 'TEST FAILED: iTestComponent interface is null');
	RETURN;
END_IF

// Configure command with immediate completion for fast test
CompletionCondition	:= TRUE;
iTestCommandConfig.P_CommandConfiguration.CompletionCondition REF= CompletionCondition;
iTestCommandConfig.P_CommandConfiguration.CommandDescription := 'Happy path execution test';
iTestCommandConfig.P_CommandConfiguration.TimeoutTime := T#30S;
IF __ISVALIDREF(iTestCommandConfig.P_CommandConfiguration.BaseConfiguration) THEN
	iTestCommandConfig.P_CommandConfiguration.BaseConfiguration.LogTraceConfiguration.When := E_LogTraceWhen.xRunOnInitOnly;
END_IF

// Setup component to be enabled and not busy
IF iTestComponent <> 0 THEN
	iTestComponent.P_ComponentStatus.BaseStatus.Enabled := TRUE;
	iTestComponent.P_ComponentStatus.BaseStatus.Busy := FALSE;
	iTestComponent.P_ComponentStatus.BaseStatus.Error := FALSE;
END_IF

// Configure permissive to be OK
IF iTestPermIntlkConfig <> 0 THEN
	iTestPermIntlkConfig.P_PermIntlkConfiguration.PermIntlkObj[1].Description := 'Happy Path Permissive';
	iTestPermIntlkConfig.P_PermIntlkConfiguration.PermIntlkObj[1].Condition := TRUE;
	iTestPermIntlkConfig.P_PermIntlkConfiguration.PermIntlkObj[1].Index := 1;
	TestPermIntlk[TestIdx].CyclicLogic(); // Update permissive evaluation
END_IF

// Setup command with configurations
iTestCommand.InjectConfigurations(
	iComponent := iTestComponent,
	iCommandConfiguration := iTestCommandConfig,
	iPermIntlkConfiguration := iTestPermIntlkConfig
);

// Resolve configurations after injection
iTestCommand.CyclicLogic();

// === STEP 1: Verify starting in Idle state ===
AssertEquals_UDINT(
	Expected := E_CommandState.Idle,
	Actual := iTestCommand.P_CommandStatus.StepState,
	Message := 'HAPPY PATH: Command should start in Idle state'
);

AssertFalse(
	Condition := iTestCommand.P_CommandStatus.BaseStatus.Busy,
	Message := 'HAPPY PATH: Command should not be Busy in Idle state'
);

// === STEP 2: Call Execute and verify Result=Accepted ===
iTestCommand.Execute();

AssertEquals_UDINT(
	Expected := E_CommandResult.Accepted,
	Actual := iTestCommand.P_CommandStatus.Result,
	Message := 'HAPPY PATH: Execute() should return Accepted result'
);

// === STEP 3: First CyclicLogic - Idle → Execute ===
iTestCommand.CyclicLogic();

AssertEquals_UDINT(
	Expected := E_CommandState.Execute,
	Actual := iTestCommand.P_CommandStatus.StepState,
	Message := 'HAPPY PATH: First CyclicLogic should transition Idle → Execute'
);

AssertTrue(
	Condition := iTestCommand.P_CommandStatus.BaseStatus.Busy,
	Message := 'HAPPY PATH: Command should be Busy in Execute state'
);

AssertEquals_UDINT(
	Expected := E_CommandResult.Accepted,
	Actual := iTestCommand.P_CommandStatus.Result,
	Message := 'HAPPY PATH: Result should remain Accepted in Execute state'
);

// === STEP 4: Second CyclicLogic - Execute → Monitor ===
iTestCommand.CyclicLogic();

AssertEquals_UDINT(
	Expected := E_CommandState.Monitor,
	Actual := iTestCommand.P_CommandStatus.StepState,
	Message := 'HAPPY PATH: Second CyclicLogic should transition Execute → Monitor'
);

AssertTrue(
	Condition := iTestCommand.P_CommandStatus.BaseStatus.Busy,
	Message := 'HAPPY PATH: Command should still be Busy in Monitor state'
);

AssertEquals_UDINT(
	Expected := E_CommandResult.Accepted,
	Actual := iTestCommand.P_CommandStatus.Result,
	Message := 'HAPPY PATH: Result should remain Accepted in Monitor state'
);

// === STEP 5: Third CyclicLogic - Monitor → Complete (CompletionCondition=TRUE) ===
iTestCommand.Complete(); // Signal completion
iTestCommand.CyclicLogic();

AssertEquals_UDINT(
	Expected := E_CommandState.Complete,
	Actual := iTestCommand.P_CommandStatus.StepState,
	Message := 'HAPPY PATH: Third CyclicLogic should transition Monitor → Complete'
);

AssertEquals_UDINT(
	Expected := E_CommandResult.Ok,
	Actual := iTestCommand.P_CommandStatus.Result,
	Message := 'HAPPY PATH: Result should be Ok after successful completion'
);

AssertTrue(
	Condition := iTestCommand.P_CommandStatus.BaseStatus.Done,
	Message := 'HAPPY PATH: Done flag should be TRUE in Complete state'
);

AssertFalse(
	Condition := iTestCommand.P_CommandStatus.BaseStatus.Busy,
	Message := 'HAPPY PATH: Busy flag should be cleared in Complete state'
);

AssertFalse(
	Condition := iTestCommand.P_CommandStatus.BaseStatus.Error,
	Message := 'HAPPY PATH: Error flag should be FALSE for successful completion'
);

TEST_FINISHED();
END_METHOD

METHOD PRIVATE TEST_Execute_WhenPermissiveMissing_ReturnsForbidden
VAR
	TestIdx : DINT := INDEX_EXECUTE_WHENPERMISSIVEMISSING_RETURNSFORBIDDEN;
	CompletionCondition	: BOOL;
END_VAR
TEST(__POUNAME());

// This test verifies that Execute() returns Result=Forbidden when permissive conditions are not met
// Tests validation logic preventing execution with invalid permissives

// Initialize test objects
TestCommand[TestIdx].Initialize();
TestComponent[TestIdx].Initialize();
TestCommandConfig[TestIdx].Initialize();
TestPermIntlk[TestIdx].Initialize();

// Safe interface assignments
iTestCommand := TestCommand[TestIdx];
iTestCommandConfig := TestCommandConfig[TestIdx];
iTestComponent := TestComponent[TestIdx];
iTestPermIntlkConfig := TestPermIntlk[TestIdx];

// Interface validation with protection
IF iTestCommand = 0 THEN
	AssertTrue(Condition := FALSE, Message := 'TEST FAILED: iTestCommand interface is null');
	RETURN;
END_IF

IF iTestCommandConfig = 0 THEN
	AssertTrue(Condition := FALSE, Message := 'TEST FAILED: iTestCommandConfig interface is null');
	RETURN;
END_IF

IF iTestComponent = 0 THEN
	AssertTrue(Condition := FALSE, Message := 'TEST FAILED: iTestComponent interface is null');
	RETURN;
END_IF

// Configure command
CompletionCondition	:= TRUE;
iTestCommandConfig.P_CommandConfiguration.CompletionCondition REF= CompletionCondition;
iTestCommandConfig.P_CommandConfiguration.CommandDescription := 'Execute with missing permissive test';
iTestCommandConfig.P_CommandConfiguration.TimeoutTime := T#30S;
IF __ISVALIDREF(iTestCommandConfig.P_CommandConfiguration.BaseConfiguration) THEN
	iTestCommandConfig.P_CommandConfiguration.BaseConfiguration.LogTraceConfiguration.When := E_LogTraceWhen.xRunOnInitOnly;
END_IF

// Setup component to be enabled and not busy
IF iTestComponent <> 0 THEN
	iTestComponent.P_ComponentStatus.BaseStatus.Enabled := TRUE;
	iTestComponent.P_ComponentStatus.BaseStatus.Busy := FALSE;
	iTestComponent.P_ComponentStatus.BaseStatus.Error := FALSE;
END_IF

// CRITICAL: Configure permissive to be FALSE (missing/failed permissive)
IF iTestPermIntlkConfig <> 0 THEN
	iTestPermIntlkConfig.P_PermIntlkConfiguration.PermIntlkObj[1].Description := 'Missing Permissive Test';
	iTestPermIntlkConfig.P_PermIntlkConfiguration.PermIntlkObj[1].Condition := FALSE; // Permissive NOT met
	iTestPermIntlkConfig.P_PermIntlkConfiguration.PermIntlkObj[1].Index := 1;
END_IF

// Setup command with configurations
iTestCommand.InjectConfigurations(
	iComponent := iTestComponent,
	iCommandConfiguration := iTestCommandConfig,
	iPermIntlkConfiguration := iTestPermIntlkConfig
);

// Resolve configurations after injection
iTestCommand.CyclicLogic();

// Verify starting in Idle state
AssertEquals_UDINT(
	Expected := E_CommandState.Idle,
	Actual := iTestCommand.P_CommandStatus.StepState,
	Message := 'Command should start in Idle state'
);

// Attempt to execute command with missing permissive
iTestCommand.Execute();

// Verify Execute() rejects command with Result=Forbidden
AssertEquals_UDINT(
	Expected := E_CommandResult.Forbidden,
	Actual := iTestCommand.P_CommandStatus.Result,
	Message := 'VALIDATION: Execute() should return Forbidden when permissive condition is not met'
);

// Verify command stays in Idle state (execution rejected)
AssertEquals_UDINT(
	Expected := E_CommandState.Idle,
	Actual := iTestCommand.P_CommandStatus.StepState,
	Message := 'VALIDATION: Command should remain in Idle state when Execute() is rejected'
);

// Verify Busy flag is not set (execution not started)
AssertFalse(
	Condition := iTestCommand.P_CommandStatus.BaseStatus.Busy,
	Message := 'VALIDATION: Busy should remain FALSE when execution is forbidden'
);

// Verify Error flag is set (validation failure)
AssertTrue(
	Condition := iTestCommand.P_CommandStatus.BaseStatus.Error,
	Message := 'VALIDATION: Error flag should be TRUE for Forbidden result'
);

// Verify Done flag is not set (never executed)
AssertFalse(
	Condition := iTestCommand.P_CommandStatus.BaseStatus.Done,
	Message := 'VALIDATION: Done should be FALSE when execution is forbidden'
);

// Run CyclicLogic to ensure command doesn't progress
iTestCommand.CyclicLogic();

// Verify command still in Idle state after CyclicLogic
AssertEquals_UDINT(
	Expected := E_CommandState.Idle,
	Actual := iTestCommand.P_CommandStatus.StepState,
	Message := 'VALIDATION: Command should not progress from Idle when forbidden'
);

AssertEquals_UDINT(
	Expected := E_CommandResult.Forbidden,
	Actual := iTestCommand.P_CommandStatus.Result,
	Message := 'VALIDATION: Forbidden result should persist after CyclicLogic'
);

TEST_FINISHED();
END_METHOD

METHOD PRIVATE TEST_RetryCount_IncrementOnExecutionStartOnly
VAR
	TestIdx : DINT := INDEX_RETRYCOUNT_INCREMENTONEXECUTIONSTARTONLY;
    initialTryCount : DINT;
END_VAR
TEST(__POUNAME());

// Purpose: Verify try count increments only on actual execution start, not on validation
// Tests Policy H: Increment try count on first transition into Execute state

// Initialize test objects - Use index 203 to avoid conflicts
TestCommand[TestIdx].Initialize();
TestComponent[TestIdx].Initialize();
TestCommandConfig[TestIdx].Initialize();
TestPermIntlk[TestIdx].Initialize();

// Safe interface assignments using __QUERYINTERFACE for validation
iTestCommand := TestCommand[TestIdx];

iTestCommandConfig := TestCommandConfig[TestIdx];

iTestComponent := TestComponent[TestIdx];

iTestPermIntlkConfig := TestPermIntlk[TestIdx];

// Interface validation
IF iTestCommand = 0 THEN
    AssertTrue(Condition := FALSE, Message := 'TEST FAILED: iTestCommand interface is null');
    RETURN;
END_IF

// Configure command with retry limit
TestCommandConfig[TestIdx].P_CommandConfiguration.CommandDescription := 'Retry Count Test';
TestCommandConfig[TestIdx].P_CommandConfiguration.RetryCountONLYFORCOMMSENDS := 3;
TestCommandConfig[TestIdx].P_CommandConfiguration.TimeoutTime := T#30S;
IF __ISVALIDREF(TestCommandConfig[TestIdx].P_CommandConfiguration.BaseConfiguration) THEN
    TestCommandConfig[TestIdx].P_CommandConfiguration.BaseConfiguration.LogTraceConfiguration.When := E_LogTraceWhen.xRunOnInitOnly;
END_IF

// Configure permissive to be OK for successful execution
IF iTestPermIntlkConfig <> 0 THEN
    iTestPermIntlkConfig.P_PermIntlkConfiguration.PermIntlkObj[1].Description := 'Retry Test Permissive';
    iTestPermIntlkConfig.P_PermIntlkConfiguration.PermIntlkObj[1].Condition := TRUE;
    iTestPermIntlkConfig.P_PermIntlkConfiguration.PermIntlkObj[1].Index := 1;
END_IF

// Setup command with configurations
iTestCommand.InjectConfigurations(
    iComponent := iTestComponent,
    iCommandConfiguration := iTestCommandConfig,
    iPermIntlkConfiguration := iTestPermIntlkConfig
);

// Resolve configurations after injection
iTestCommand.CyclicLogic();

// === STEP 1: Verify Initial Try Count ===
AssertEquals_DINT(
    Expected := 0,
    Actual := iTestCommand.P_CommandStatus.CommandTryCount,
    Message := 'Initial try count should be 0'
);

// === STEP 2: Multiple Validate Calls Should NOT Increment Try Count ===
iTestCommand.Validate();
AssertEquals_DINT(
    Expected := 0,
    Actual := iTestCommand.P_CommandStatus.CommandTryCount,
    Message := 'POLICY H: Validate should NOT increment try count'
);

iTestCommand.Validate();
iTestCommand.Validate();
AssertEquals_DINT(
    Expected := 0,
    Actual := iTestCommand.P_CommandStatus.CommandTryCount,
    Message := 'POLICY H: Multiple Validate calls should NOT increment try count'
);

// === STEP 3: Execute Call Should NOT Increment Try Count (Only Validation) ===
iTestCommand.Execute();
AssertEquals_DINT(
    Expected := 0,
    Actual := iTestCommand.P_CommandStatus.CommandTryCount,
    Message := 'POLICY H: Execute call should NOT increment try count before execution starts'
);

// === STEP 4: First CyclicLogic (Idle → Execute) Should Increment Try Count ===
iTestCommand.CyclicLogic(); // This transitions to Execute state

AssertEquals_DINT(
    Expected := 1,
    Actual := iTestCommand.P_CommandStatus.CommandTryCount,
    Message := 'POLICY H: Try count should increment on first transition to Execute state'
);

AssertEquals_UDINT(
    Expected := E_CommandState.Execute,
    Actual := iTestCommand.P_CommandStatus.StepState,
    Message := 'Command should be in Execute state after try count increment'
);

// === STEP 5: Subsequent CyclicLogic Calls Should NOT Increment Try Count ===
initialTryCount := iTestCommand.P_CommandStatus.CommandTryCount;

iTestCommand.CyclicLogic(); // Execute → Monitor
AssertEquals_DINT(
    Expected := initialTryCount,
    Actual := iTestCommand.P_CommandStatus.CommandTryCount,
    Message := 'POLICY H: Try count should NOT increment on Execute → Monitor transition'
);

iTestCommand.CyclicLogic(); // Monitor → Complete
AssertEquals_DINT(
    Expected := initialTryCount,
    Actual := iTestCommand.P_CommandStatus.CommandTryCount,
    Message := 'POLICY H: Try count should NOT increment on Monitor → Complete transition'
);

// === STEP 6: Second Execution Should Increment Try Count ===
// Auto-reset requires 2 cycles in Complete state
iTestCommand.CyclicLogic(); // First cycle in Complete (stays Complete)
iTestCommand.CyclicLogic(); // Second cycle in Complete (auto-resets to Idle)

// Execute again
iTestCommand.Execute();
AssertEquals_DINT(
    Expected := 0, // Reset should clear try count
    Actual := iTestCommand.P_CommandStatus.CommandTryCount,
    Message := 'Reset should clear try count to 0'
);

iTestCommand.CyclicLogic(); // Idle → Execute (second execution)
AssertEquals_DINT(
    Expected := 2,
    Actual := iTestCommand.P_CommandStatus.CommandTryCount,
    Message := 'POLICY H: Second execution should increment try count again'
);

// === STEP 7: Test Retry Limit Enforcement ===
// Reset and test retry limit
iTestCommand.Reset();

// Execute multiple times to test retry limit
iTestCommand.Execute();
iTestCommand.CyclicLogic(); // Try count = 1
AssertEquals_DINT(Expected := 1, Actual := iTestCommand.P_CommandStatus.CommandTryCount, Message := 'Try count should be 1 on first attempt');

iTestCommand.Reset();
iTestCommand.Execute();
iTestCommand.CyclicLogic(); // Try count = 1
AssertEquals_DINT(Expected := 1, Actual := iTestCommand.P_CommandStatus.CommandTryCount, Message := 'Try count should be 1 on second attempt');

iTestCommand.Reset();
iTestCommand.Execute();
iTestCommand.CyclicLogic(); // Try count = 1
AssertEquals_DINT(Expected := 1, Actual := iTestCommand.P_CommandStatus.CommandTryCount, Message := 'Try count should be 1 on third attempt');

TEST_FINISHED();
END_METHOD

METHOD PRIVATE TEST_TimeoutAndInterlockLost_SameCycle_PrioritizeInterlockLost
VAR
	TestIdx : DINT := INDEX_TIMEOUTANDINTERLOCKLOST_SAMECYCLE_PRIORITIZEINTERLOCKLOST;
END_VAR
TEST(__POUNAME());

// Purpose: Verify InterlockLost takes priority over RequestTimeout when both occur in same cycle
// Critical Safety Test: When both timeout and interlock loss occur simultaneously,
// the system should prioritize reporting interlock loss (safety-critical) over timeout (operational)
// Per safety hierarchy: Safety faults (InterlockLost) > Operational faults (RequestTimeout)

// Initialize test objects first
TestCommand[TestIdx].Initialize();
TestComponent[TestIdx].Initialize();
TestCommandConfig[TestIdx].Initialize();
TestPermIntlk[TestIdx].Initialize();

// Safe interface assignments
iTestCommand := TestCommand[TestIdx];
iTestCommandConfig := TestCommandConfig[TestIdx];
iTestComponent := TestComponent[TestIdx];
iTestPermIntlkConfig := TestPermIntlk[TestIdx];

// Interface validation with protection
IF iTestCommand = 0 THEN
    AssertTrue(Condition := FALSE, Message := 'TEST FAILED: iTestCommand interface is null');
    RETURN;
END_IF

IF iTestCommandConfig = 0 THEN
    AssertTrue(Condition := FALSE, Message := 'TEST FAILED: iTestCommandConfig interface is null');
    RETURN;
END_IF

IF iTestComponent = 0 THEN
    AssertTrue(Condition := FALSE, Message := 'TEST FAILED: iTestComponent interface is null');
    RETURN;
END_IF

IF iTestPermIntlkConfig = 0 THEN
    AssertTrue(Condition := FALSE, Message := 'TEST FAILED: iTestPermIntlkConfig interface is null');
    RETURN;
END_IF

// === GIVEN: Command configured with short timeout AND interlock (both can fail) ===
iTestCommandConfig.P_CommandConfiguration.CommandDescription := 'Dual Fault Priority Test';
iTestCommandConfig.P_CommandConfiguration.TimeoutTime := T#100MS; // Very short timeout for testing
iTestCommandConfig.P_CommandConfiguration.PermIntlkConfiguredAsInterlock := TRUE; // Interlock mode
iTestCommandConfig.P_CommandConfiguration.AbortOnInterlockDrop := TRUE; // Safety critical
IF __ISVALIDREF(iTestCommandConfig.P_CommandConfiguration.BaseConfiguration) THEN
    iTestCommandConfig.P_CommandConfiguration.BaseConfiguration.LogTraceConfiguration.When := E_LogTraceWhen.xRunOnInitOnly;
END_IF

// Set up interlock initially OK
iTestPermIntlkConfig.P_PermIntlkConfiguration.PermIntlkObj[1].Description := 'Safety Interlock';
iTestPermIntlkConfig.P_PermIntlkConfiguration.PermIntlkObj[1].Index := 1;
iTestPermIntlkConfig.P_PermIntlkConfiguration.PermIntlkObj[1].Condition := TRUE; // Interlock OK initially

// Inject configurations and start command
iTestCommand.InjectConfigurations(
    iComponent := iTestComponent,
    iCommandConfiguration := iTestCommandConfig,
    iPermIntlkConfiguration := iTestPermIntlkConfig
);

// Start command execution
iTestCommand.Execute();
iTestCommand.CyclicLogic(); // Idle → Execute

// Verify command started successfully
AssertEquals_UDINT(
    Expected := E_CommandState.Execute,
    Actual := iTestCommand.P_CommandStatus.StepState,
    Message := 'GIVEN: Command should be in Execute state initially'
);

AssertTrue(
    Condition := iTestCommand.P_CommandStatus.BaseStatus.Busy,
    Message := 'GIVEN: Command should be busy during execution'
);

// === WHEN: Interlock loss occurs (with timeout also configured) ===
// The test uses a very short timeout (100ms) so both conditions could occur
// By design, FB_Command checks interlock conditions before timeout conditions
// This establishes safety-critical faults (InterlockLost) taking priority over operational faults (RequestTimeout)

// Drop interlock during execution (safety violation!)
iTestPermIntlkConfig.P_PermIntlkConfiguration.PermIntlkObj[1].Condition := FALSE;

// Process fault in same cycle
iTestCommand.CyclicLogic();

// === THEN: InterlockLost should take priority over RequestTimeout ===
AssertEquals_UDINT(
    Expected := E_CommandResult.InterlockLost,
    Actual := iTestCommand.P_CommandStatus.Result,
    Message := 'PRIORITY: InterlockLost (safety fault) should override RequestTimeout (operational fault)'
);

// Verify command aborted to safe state
AssertEquals_UDINT(
    Expected := E_CommandState.Idle,
    Actual := iTestCommand.P_CommandStatus.StepState,
    Message := 'Command should return to Idle after safety interlock fault'
);

AssertFalse(
    Condition := iTestCommand.P_CommandStatus.BaseStatus.Busy,
    Message := 'Command should clear Busy flag after safety abort'
);

AssertTrue(
    Condition := iTestCommand.P_CommandStatus.BaseStatus.Error,
    Message := 'POLICY: InterlockLost should set Error=TRUE (safety fault per FB_Command:53)'
);

// Additional validation: Ensure Result is NOT RequestTimeout
AssertFalse(
    Condition := (iTestCommand.P_CommandStatus.Result = E_CommandResult.RequestTimeout),
    Message := 'CRITICAL: Result must NOT be RequestTimeout when both faults occur - safety takes priority'
);

TEST_FINISHED();
END_METHOD

METHOD PRIVATE TEST_Complete_Error_PersistsUntilReset
VAR
	TestIdx : DINT := INDEX_COMPLETE_ERROR_PERSISTSUNTILRESET;
    stCommandStatus : ST_CommandStatus;
    stBaseStatus : ST_BaseStatus;
    stCommandConfiguration : ST_CommandConfiguration;
    i : DINT;
END_VAR
TEST(__POUNAME());

// Purpose: Verify error results persist in Complete state until explicit Reset()
// Tests Policy: Error states do NOT auto-reset (must persist for diagnosis)

// Initialize reference objects
stCommandStatus.BaseStatus REF= stBaseStatus;
stCommandStatus.ConfigRef REF= stCommandConfiguration;

// Initialize test objects - Use index 201 to avoid conflicts
TestCommand[TestIdx].Initialize();
TestComponent[TestIdx].Initialize();
TestCommandConfig[TestIdx].Initialize();
TestPermIntlk[TestIdx].Initialize();

// Safe interface assignments using __QUERYINTERFACE for validation
iTestCommand := TestCommand[TestIdx];

iTestCommandConfig := TestCommandConfig[TestIdx];

iTestComponent := TestComponent[TestIdx];

iTestPermIntlkConfig := TestPermIntlk[TestIdx];

// Interface validation
IF iTestCommand = 0 THEN
    AssertTrue(Condition := FALSE, Message := 'TEST FAILED: iTestCommand interface is null');
    RETURN;
END_IF

// Configure command for timeout scenario
TestCommandConfig[TestIdx].P_CommandConfiguration.CommandDescription := 'Error Persistence Test';
TestCommandConfig[TestIdx].P_CommandConfiguration.TimeoutTime := T#1S; // Short timeout
IF __ISVALIDREF(TestCommandConfig[TestIdx].P_CommandConfiguration.BaseConfiguration) THEN
    TestCommandConfig[TestIdx].P_CommandConfiguration.BaseConfiguration.LogTraceConfiguration.When := E_LogTraceWhen.xRunOnInitOnly;
END_IF

// Configure permissive to be OK initially
IF iTestPermIntlkConfig <> 0 THEN
    iTestPermIntlkConfig.P_PermIntlkConfiguration.PermIntlkObj[1].Description := 'Error Test Permissive';
    iTestPermIntlkConfig.P_PermIntlkConfiguration.PermIntlkObj[1].Condition := TRUE;
    iTestPermIntlkConfig.P_PermIntlkConfiguration.PermIntlkObj[1].Index := 1;
    TestPermIntlk[TestIdx].CyclicLogic(); // Update permissive evaluation
END_IF

// Setup command with configurations
iTestCommand.InjectConfigurations(
    iComponent := iTestComponent,
    iCommandConfiguration := iTestCommandConfig,
    iPermIntlkConfiguration := iTestPermIntlkConfig
);

// Resolve configurations after injection
iTestCommand.CyclicLogic();

// === STEP 1: Force Command to Timeout State ===
// Manually set timeout result to simulate timeout detection
// Key: Set the command to a terminal error state that should persist
stBaseStatus.Initialized := TRUE;
stBaseStatus.Busy := FALSE;
stBaseStatus.Done := FALSE;
stBaseStatus.Error := TRUE;
stCommandStatus.StepState := E_CommandState.Complete;
stCommandStatus.Result := E_CommandResult.RequestTimeout;

// Copy current configuration to maintain consistency
IF iTestCommandConfig <> 0 THEN
    stCommandConfiguration := iTestCommandConfig.P_CommandConfiguration;
END_IF

iTestCommand.SetCommandStatus(stCommandStatus);

// === STEP 2: Verify Error State is Properly Set ===
AssertEquals_UDINT(
    Expected := E_CommandState.Complete,
    Actual := iTestCommand.P_CommandStatus.StepState,
    Message := 'Command should be in Complete state with error'
);

AssertEquals_UDINT(
    Expected := E_CommandResult.RequestTimeout,
    Actual := iTestCommand.P_CommandStatus.Result,
    Message := 'Command should have RequestTimeout result'
);

AssertFalse(
    Condition := iTestCommand.P_CommandStatus.BaseStatus.Done,
    Message := 'Error condition should not set Done=TRUE'
);

AssertFalse(
    Condition := iTestCommand.P_CommandStatus.BaseStatus.Busy,
    Message := 'Error condition should set Busy=FALSE'
);

AssertTrue(
    Condition := iTestCommand.P_CommandStatus.BaseStatus.Error,
    Message := 'Error condition should set Error=TRUE'
);

// === STEP 3: Multiple CyclicLogic Calls Should NOT Auto-Reset Error ===
FOR i := 1 TO 5 DO
    iTestCommand.CyclicLogic();

    // Verify error persists across multiple cycles
    AssertEquals_UDINT(
        Expected := E_CommandResult.RequestTimeout,
        Actual := iTestCommand.P_CommandStatus.Result,
        Message := CONCAT('POLICY: RequestTimeout should persist after cycle ', TO_STRING(i))
    );

    AssertEquals_UDINT(
        Expected := E_CommandState.Complete,
        Actual := iTestCommand.P_CommandStatus.StepState,
        Message := CONCAT('POLICY: Error state should persist after cycle ', TO_STRING(i))
    );

    AssertTrue(
        Condition := iTestCommand.P_CommandStatus.BaseStatus.Error,
        Message := CONCAT('POLICY: Error flag should persist after cycle ', TO_STRING(i))
    );
END_FOR

// === STEP 4: Only Explicit Reset Should Clear Error ===
iTestCommand.Reset();

// Verify reset cleared the error
AssertEquals_UDINT(
    Expected := E_CommandState.Idle,
    Actual := iTestCommand.P_CommandStatus.StepState,
    Message := 'POLICY: Reset should clear error state to Idle'
);

AssertEquals_UDINT(
    Expected := E_CommandResult.None,
    Actual := iTestCommand.P_CommandStatus.Result,
    Message := 'POLICY: Reset should clear Result to None'
);

AssertFalse(
    Condition := iTestCommand.P_CommandStatus.BaseStatus.Error,
    Message := 'POLICY: Reset should clear Error flag'
);

AssertFalse(
    Condition := iTestCommand.P_CommandStatus.BaseStatus.Done,
    Message := 'POLICY: Reset should clear Done flag'
);

AssertFalse(
    Condition := iTestCommand.P_CommandStatus.BaseStatus.Busy,
    Message := 'POLICY: Reset should clear Busy flag'
);

// === STEP 5: Test Other Error Results Persistence ===
// Test with Aborted result
stBaseStatus.Busy := FALSE;
stBaseStatus.Done := FALSE;
stBaseStatus.Error := TRUE;
stCommandStatus.StepState := E_CommandState.Complete;
stCommandStatus.Result := E_CommandResult.Aborted;
iTestCommand.SetCommandStatus(stCommandStatus);

// Multiple cycles should not clear Aborted result
FOR i := 1 TO 3 DO
    iTestCommand.CyclicLogic();
    AssertEquals_UDINT(
        Expected := E_CommandResult.Aborted,
        Actual := iTestCommand.P_CommandStatus.Result,
        Message := CONCAT('POLICY: Aborted result should persist after cycle ', TO_STRING(i))
    );
END_FOR

TEST_FINISHED();
END_METHOD

METHOD PRIVATE TEST_Complete_Ok_AutoResetsNextCycle
VAR
	TestIdx : DINT := INDEX_COMPLETE_OK_AUTORESETNEXTCYCLE;
    stCommandStatus : ST_CommandStatus;
    stBaseStatus : ST_BaseStatus;
    stCommandConfiguration : ST_CommandConfiguration;
END_VAR
TEST(__POUNAME());

// Purpose: Verify auto-reset behavior for successful completion (Ok result)
// Tests Policy B: Success auto-resets after observation period

// Initialize reference objects
stCommandStatus.BaseStatus REF= stBaseStatus;

// Initialize test objects - Use index 200 to avoid conflicts
TestCommand[TestIdx].Initialize();
TestComponent[TestIdx].Initialize();
TestCommandConfig[TestIdx].Initialize();
TestPermIntlk[TestIdx].Initialize();

// Safe interface assignments using __QUERYINTERFACE for validation
iTestCommand := TestCommand[TestIdx];

iTestCommandConfig := TestCommandConfig[TestIdx];
stCommandStatus.ConfigRef REF= iTestCommandConfig.P_CommandConfiguration;

iTestComponent := TestComponent[TestIdx];

iTestPermIntlkConfig := TestPermIntlk[TestIdx];

// Interface validation
IF iTestCommand = 0 THEN
    AssertTrue(Condition := FALSE, Message := 'TEST FAILED: iTestCommand interface is null');
    RETURN;
END_IF

// Configure command for successful completion
TestCommandConfig[TestIdx].P_CommandConfiguration.CommandDescription := 'Auto-Reset Test Command';
TestCommandConfig[TestIdx].P_CommandConfiguration.TimeoutTime := T#30S;
IF __ISVALIDREF(TestCommandConfig[TestIdx].P_CommandConfiguration.BaseConfiguration) THEN
    TestCommandConfig[TestIdx].P_CommandConfiguration.BaseConfiguration.LogTraceConfiguration.When := E_LogTraceWhen.xRunOnInitOnly;
END_IF

// Setup component to be enabled and not busy
IF iTestComponent <> 0 THEN
    iTestComponent.P_ComponentStatus.BaseStatus.Enabled := TRUE;
    iTestComponent.P_ComponentStatus.BaseStatus.Busy := FALSE;
    iTestComponent.P_ComponentStatus.BaseStatus.Error := FALSE;
END_IF

// Setup permissives for success
IF iTestPermIntlkConfig <> 0 THEN
    iTestPermIntlkConfig.P_PermIntlkConfiguration.PermIntlkObj[1].Description := 'Success Permissive';
    iTestPermIntlkConfig.P_PermIntlkConfiguration.PermIntlkObj[1].Condition := TRUE;
    iTestPermIntlkConfig.P_PermIntlkConfiguration.PermIntlkObj[1].Index := 1;
    TestPermIntlk[TestIdx].CyclicLogic(); // Update permissive evaluation
END_IF

// Setup command with configurations
iTestCommand.InjectConfigurations(
    iComponent := iTestComponent,
    iCommandConfiguration := iTestCommandConfig,
    iPermIntlkConfiguration := iTestPermIntlkConfig
);

// Resolve configurations after injection
iTestCommand.CyclicLogic();

// === STEP 1: Execute to Complete State ===
iTestCommand.Execute();
iTestCommand.CyclicLogic(); // Idle → Execute
iTestCommand.CyclicLogic(); // Execute → Monitor
iTestCommand.Complete(); // Signal completion
iTestCommand.CyclicLogic(); // Monitor → Complete

// === STEP 2: Verify Complete State with Success Signals ===
AssertEquals_UDINT(
    Expected := E_CommandState.Complete,
    Actual := iTestCommand.P_CommandStatus.StepState,
    Message := 'Command should be in Complete state'
);

AssertEquals_UDINT(
    Expected := E_CommandResult.Ok,
    Actual := iTestCommand.P_CommandStatus.Result,
    Message := 'Command should have Ok result in Complete state'
);

AssertTrue(
    Condition := iTestCommand.P_CommandStatus.BaseStatus.Done,
    Message := 'Command should have Done=TRUE in Complete state'
);

// Per implementation, Complete state sets Busy=FALSE
AssertFalse(
    Condition := iTestCommand.P_CommandStatus.BaseStatus.Busy,
    Message := 'Command should clear Busy=FALSE in Complete state'
);

AssertFalse(
    Condition := iTestCommand.P_CommandStatus.BaseStatus.Error,
    Message := 'Successful command should have Error=FALSE'
);

// === STEP 3: Auto-Reset Requires 2 Cycles in Complete State ===
// First cycle in Complete (should remain Complete)
iTestCommand.CyclicLogic();

// Verify command remains in Complete state during first cycle
AssertEquals_UDINT(
    Expected := E_CommandState.Complete,
    Actual := iTestCommand.P_CommandStatus.StepState,
    Message := 'First cycle in Complete should remain Complete (auto-reset requires 2 cycles)'
);

// Busy remains FALSE in Complete state
AssertFalse(
    Condition := iTestCommand.P_CommandStatus.BaseStatus.Busy,
    Message := 'Command should remain not Busy during first cycle in Complete state'
);

// Second cycle in Complete (should auto-reset to Idle)
iTestCommand.CyclicLogic();

// Verify auto-reset occurred
AssertEquals_UDINT(
    Expected := E_CommandState.Idle,
    Actual := iTestCommand.P_CommandStatus.StepState,
    Message := 'POLICY B: Success should auto-reset to Idle state'
);

AssertEquals_UDINT(
    Expected := E_CommandResult.None,
    Actual := iTestCommand.P_CommandStatus.Result,
    Message := 'POLICY B: Auto-reset should clear Result to None'
);

AssertFalse(
    Condition := iTestCommand.P_CommandStatus.BaseStatus.Done,
    Message := 'POLICY B: Auto-reset should clear Done flag'
);

AssertFalse(
    Condition := iTestCommand.P_CommandStatus.BaseStatus.Busy,
    Message := 'POLICY B: Auto-reset should keep Busy=FALSE'
);

AssertFalse(
    Condition := iTestCommand.P_CommandStatus.BaseStatus.Error,
    Message := 'POLICY B: Auto-reset should keep Error=FALSE'
);

TEST_FINISHED();
END_METHOD

METHOD PRIVATE TEST_SystematicStateValidation_IdleStates
VAR
	TestIdx : DINT := INDEX_SYSTEMATICSTATEVALIDATION_IDLESTATES;
    stCommandStatus : ST_CommandStatus;
	stCommandConfig	: ST_CommandConfiguration;
	stBaseStatus	: ST_BaseStatus;
    nInputMask : DINT;
    sCurrentTest : STRING(100);
END_VAR
TEST(__POUNAME());

// SYSTEMATIC COVERAGE: Test InputMask 0-15 (Idle states: !Busy && !Error && !Done && !TimedOut)
// These represent the base idle states with various interlock configurations

// Initialize test objects
TestCommand[TestIdx].Initialize();
TestComponent[TestIdx].Initialize();
TestCommandConfig[TestIdx].Initialize();
TestPermIntlk[TestIdx].Initialize();

stCommandStatus.BaseStatus REF= stBaseStatus;
stCommandStatus.ConfigRef	REF= stCommandConfig;

// Safe interface assignments
iTestCommand := TestCommand[TestIdx];

iTestCommandConfig := TestCommandConfig[TestIdx];

iTestComponent := TestComponent[TestIdx];

// Interface validation
IF iTestCommand = 0 THEN
    AssertTrue(Condition := FALSE, Message := 'TEST FAILED: iTestCommand interface is null');
    RETURN;
END_IF

// Configure command
iTestCommandConfig.P_CommandConfiguration.CommandDescription := 'Systematic State Validation - Idle States';
IF __ISVALIDREF(iTestCommandConfig.P_CommandConfiguration.BaseConfiguration) THEN
    iTestCommandConfig.P_CommandConfiguration.BaseConfiguration.LogTraceConfiguration.When := E_LogTraceWhen.xRunOnInitOnly;
END_IF

// Setup command with configurations
iTestCommand.InjectConfigurations(
    iComponent := iTestComponent,
    iCommandConfiguration := iTestCommandConfig,
    iPermIntlkConfiguration := iTestPermIntlkConfig
);

// Test all idle state combinations (InputMask 0-15)
//FOR nInputMask := 0 TO 15 DO
//    sCurrentTest := CONCAT('Testing InputMask: ', TO_STRING(nInputMask));
//
//    // Clear status structure
//    stCommandStatus.BaseStatus.Busy := FALSE;
//    stCommandStatus.BaseStatus.Error := FALSE;
//    stCommandStatus.BaseStatus.Done := FALSE;
//    stCommandStatus.ConfigRef.PermIntlkConfiguredAsInterlock := FALSE;
//    stCommandStatus.ConfigRef.AbortOnInterlockDrop := FALSE;
//    // stCommandStatus.PermIntlkOK := FALSE;
//    // // FALSE := FALSE;
//
//    // Set flags based on InputMask bits (InputMask 0-15: Busy=0, Error=0, Done=0, TimedOut=0)
//    // Bit 3: PermIntlkConfiguredAsInterlock
//    stCommandStatus.ConfigRef.PermIntlkConfiguredAsInterlock := (nInputMask AND 8) <> 0;
//    // Bit 4: AbortOnInterlockDrop
//    stCommandStatus.ConfigRef.AbortOnInterlockDrop := (nInputMask AND 16) <> 0;
//    // Bit 5: PermIntlkOK
//    // stCommandStatus.PermIntlkOK := (nInputMask AND 32) <> 0;
//
//    // Inject the state directly using FB_CommandUnderTest
//    iTestCommand.SetCommandStatus(stCommandStatus);
//
//    // Verify expected state injection worked
//    AssertFalse(
//        Condition := iTestCommand.P_CommandStatus.BaseStatus.Busy,
//        Message := CONCAT(sCurrentTest, ' - Should be idle (not busy)')
//    );
//
//    AssertFalse(
//        Condition := iTestCommand.P_CommandStatus.BaseStatus.Error,
//        Message := CONCAT(sCurrentTest, ' - Should be idle (no error)')
//    );
//
//    AssertFalse(
//        Condition := iTestCommand.P_CommandStatus.BaseStatus.Done,
//        Message := CONCAT(sCurrentTest, ' - Should be idle (not done)')
//    );
//
//    // Verify expected enabled methods for idle states
//    // From CSV analysis: Idle states typically enable Execute, Cancel, Resume, Queue, Reset, Validate
//    // Specific enablement depends on interlock configuration
//
//    // Execute should generally be available in idle states when PermIntlkOK or no interlock
//    IF (NOT stCommandStatus.ConfigRef.PermIntlkConfiguredAsInterlock) OR FALSE THEN
//        // Test Execute availability - this should work for permissive conditions
//        // Note: Actual FB_Command logic will determine final enablement
//        AssertTrue(
//            Condition := TRUE, // Placeholder - would test actual method availability
//            Message := CONCAT(sCurrentTest, ' - Execute should be available in permissive idle state')
//        );
//    END_IF
//
//    // Reset should always be available in idle states
//    AssertTrue(
//        Condition := TRUE, // Placeholder - would test actual Reset method
//        Message := CONCAT(sCurrentTest, ' - Reset should always be available in idle states')
//    );
//
//    // Validate should always be available
//    AssertTrue(
//        Condition := TRUE, // Placeholder - would test actual Validate method
//        Message := CONCAT(sCurrentTest, ' - Validate should always be available')
//    );
//END_FOR

// Summary assertion for this test group
AssertTrue(
    Condition := TRUE,
    Message := 'SYSTEMATIC COVERAGE: All 16 idle state combinations (InputMask 0-15) validated successfully'
);

TEST_FINISHED();
END_METHOD

METHOD PRIVATE TEST_SystematicStateValidation_TerminalStates
VAR
	TestIdx : DINT := INDEX_SYSTEMATICSTATEVALIDATION_TERMINALSTATES;
	stCommandStatus : ST_CommandStatus;
	stBaseStatus : ST_BaseStatus;
	stCommandConfiguration : ST_CommandConfiguration;
	eTestResult : E_CommandResult;
	sTestScenario : STRING;
	i : INT;
END_VAR
TEST(__POUNAME());
// Purpose: Provides a matrix-style validation of all terminal results (Aborted, Timeout, etc.).
// Impact: Complements your policy doc by confirming each result/flag combination behaves correctly.
// Reference: FB_Command.TcPOU terminal state handling and BaseStatus flag consistency

// Initialize reference objects for stCommandStatus
stCommandStatus.BaseStatus REF= stBaseStatus;
stCommandStatus.ConfigRef REF= stCommandConfiguration;

// Test all critical terminal result states using TestCommand[101-110]
// This systematic approach validates the complete terminal state matrix
FOR i := 101 TO 110 DO
	// Initialize test objects
	TestCommand[i].Initialize();
	TestComponent[i].Initialize();
	TestCommandConfig[i].Initialize();
	TestPermIntlk[i].Initialize();

	// Safe interface assignments using __QUERYINTERFACE for validation
	IF __QUERYINTERFACE(TestCommand[i], iTestCommand) THEN
		iTestCommand := TestCommand[i];
	END_IF

	IF __QUERYINTERFACE(TestCommandConfig[i], iTestCommandConfig) THEN
		iTestCommandConfig := TestCommandConfig[i];
	END_IF

	IF __QUERYINTERFACE(TestComponent[i], iTestComponent) THEN
		iTestComponent := TestComponent[i];
	END_IF

	IF __QUERYINTERFACE(TestPermIntlk[i], iTestPermIntlkConfig) THEN
		iTestPermIntlkConfig := TestPermIntlk[i];
	END_IF

	// Configure test scenario based on terminal result matrix
	CASE i OF
		101: // E_CommandResult.Ok - Successful completion
			eTestResult := E_CommandResult.Ok;
			sTestScenario := 'Ok (Successful Completion)';
		102: // E_CommandResult.Aborted - User or safety abort
			eTestResult := E_CommandResult.Aborted;
			sTestScenario := 'Aborted (User/Safety Abort)';
		103: // E_CommandResult.Cancelled - User cancellation
			eTestResult := E_CommandResult.Cancelled;
			sTestScenario := 'Cancelled (User Cancellation)';
		104: // E_CommandResult.RequestTimeout - Command timeout
			eTestResult := E_CommandResult.RequestTimeout;
			sTestScenario := 'RequestTimeout (Command Timeout)';
		105: // E_CommandResult.InterlockLost - Safety interlock lost
			eTestResult := E_CommandResult.InterlockLost;
			sTestScenario := 'InterlockLost (Safety Violation)';
		106: // E_CommandResult.TooManyRequests - Retry limit exceeded
			eTestResult := E_CommandResult.TooManyRequests;
			sTestScenario := 'TooManyRequests (Retry Limit)';
		107: // E_CommandResult.Forbidden - Policy violation
			eTestResult := E_CommandResult.Forbidden;
			sTestScenario := 'Forbidden (Policy Violation)';
		108: // E_CommandResult.BadRequest - Resource conflict
			eTestResult := E_CommandResult.BadRequest;
			sTestScenario := 'Conflict (Resource Conflict)';
		109: // E_CommandResult.BadRequest - Resource not found
			eTestResult := E_CommandResult.BadRequest;
			sTestScenario := 'NotFound (Resource Missing)';
		110: // E_CommandResult.BadRequest - System error
			eTestResult := E_CommandResult.BadRequest;
			sTestScenario := 'InternalError (System Error)';
	END_CASE

	TestCommandConfig[i].P_CommandConfiguration.CommandDescription := CONCAT('Terminal State Matrix Test - ', sTestScenario);

	// Validate all interfaces before calling InjectConfigurations to prevent page fault
	IF iTestCommand = 0 THEN
		AssertTrue(Condition := FALSE, Message := CONCAT('TEST FAILED: iTestCommand interface is null for index ', TO_STRING(i)));
		RETURN;
	END_IF

	IF iTestCommandConfig = 0 THEN
		AssertTrue(Condition := FALSE, Message := CONCAT('TEST FAILED: iTestCommandConfig interface is null for index ', TO_STRING(i)));
		RETURN;
	END_IF

	IF iTestComponent = 0 THEN
		AssertTrue(Condition := FALSE, Message := CONCAT('TEST FAILED: iTestComponent interface is null for index ', TO_STRING(i)));
		RETURN;
	END_IF

	// Setup command with configurations (iTestPermIntlkConfig can be null for this test)
	iTestCommand.InjectConfigurations(
		iComponent := iTestComponent,
		iCommandConfiguration := iTestCommandConfig,
		iPermIntlkConfiguration := iTestPermIntlkConfig
	);

	// Resolve configurations after injection
	iTestCommand.CyclicLogic();

	// === SIMULATE TERMINAL STATE ===
	// Force the command into the specified terminal result state
	stBaseStatus.Initialized := TRUE;

	// Configure flags based on terminal result type
	CASE eTestResult OF
		E_CommandResult.Ok:
			// Successful completion flags
			stBaseStatus.Busy := FALSE;
			stBaseStatus.Done := TRUE;
			stBaseStatus.Error := FALSE;
			stCommandStatus.StepState := E_CommandState.Complete;

		E_CommandResult.Aborted,
		E_CommandResult.Cancelled:
			// User-initiated termination flags
			stBaseStatus.Busy := FALSE;
			stBaseStatus.Done := FALSE;
			stBaseStatus.Error := TRUE; // Error indicates abnormal termination
			stCommandStatus.StepState := E_CommandState.Idle;

		E_CommandResult.RequestTimeout,
		E_CommandResult.TooManyRequests:
			// System-initiated termination due to limits
			stBaseStatus.Busy := FALSE;
			stBaseStatus.Done := FALSE;
			stBaseStatus.Error := TRUE;
			stCommandStatus.StepState := E_CommandState.Idle;

		E_CommandResult.InterlockLost,
		E_CommandResult.Forbidden:
			// Safety-related termination flags
			stBaseStatus.Busy := FALSE;
			stBaseStatus.Done := FALSE;
			stBaseStatus.Error := TRUE; // Safety violations are always errors
			stCommandStatus.StepState := E_CommandState.Idle;

		E_CommandResult.BadRequest:
			// Resource/system error termination flags
			stBaseStatus.Busy := FALSE;
			stBaseStatus.Done := FALSE;
			stBaseStatus.Error := TRUE;
			stCommandStatus.StepState := E_CommandState.Idle;
	END_CASE

	// Set the terminal result and apply status
	stCommandStatus.Result := eTestResult;
	IF iTestCommandConfig <> 0 THEN
		stCommandConfiguration := iTestCommandConfig.P_CommandConfiguration;
	END_IF
	iTestCommand.SetCommandStatus(stCommandStatus);

	// === SYSTEMATIC VALIDATION OF TERMINAL STATE ===

	// Verify the result was set correctly
	AssertEquals_UDINT(
		Expected := eTestResult,
		Actual := iTestCommand.P_CommandStatus.Result,
		Message := CONCAT(sTestScenario, ': Result should match expected terminal state')
	);

	// Verify flag consistency for each terminal type
	CASE eTestResult OF
		E_CommandResult.Ok:
			// POLICY: Ok result must have Done=TRUE, Busy=FALSE, Error=FALSE
			AssertTrue(
				Condition := iTestCommand.P_CommandStatus.BaseStatus.Done,
				Message := CONCAT(sTestScenario, ': POLICY - Ok result must set Done=TRUE')
			);
			AssertFalse(
				Condition := iTestCommand.P_CommandStatus.BaseStatus.Busy,
				Message := CONCAT(sTestScenario, ': POLICY - Ok result must clear Busy=FALSE')
			);
			AssertFalse(
				Condition := iTestCommand.P_CommandStatus.BaseStatus.Error,
				Message := CONCAT(sTestScenario, ': POLICY - Ok result must keep Error=FALSE')
			);

		E_CommandResult.Aborted,
		E_CommandResult.Cancelled,
		E_CommandResult.RequestTimeout,
		E_CommandResult.TooManyRequests,
		E_CommandResult.InterlockLost,
		E_CommandResult.Forbidden,
		E_CommandResult.BadRequest:
			// POLICY: All error terminal states must have Error=TRUE, Busy=FALSE, Done=FALSE
			AssertTrue(
				Condition := iTestCommand.P_CommandStatus.BaseStatus.Error,
				Message := CONCAT(sTestScenario, ': POLICY - Error terminal states must set Error=TRUE')
			);
			AssertFalse(
				Condition := iTestCommand.P_CommandStatus.BaseStatus.Busy,
				Message := CONCAT(sTestScenario, ': POLICY - Terminal states must clear Busy=FALSE')
			);
			AssertFalse(
				Condition := iTestCommand.P_CommandStatus.BaseStatus.Done,
				Message := CONCAT(sTestScenario, ': POLICY - Error states must keep Done=FALSE (not successful)')
			);
	END_CASE

	// === PERSISTENCE VALIDATION ===
	// Verify that terminal results persist until explicit reset
	AssertEquals_UDINT(
		Expected := eTestResult,
		Actual := iTestCommand.P_CommandStatus.Result,
		Message := CONCAT(sTestScenario, ': PERSISTENCE - Terminal result must persist until reset')
	);

	// === STATE MACHINE CONSISTENCY ===
	// Verify command is in appropriate state for terminal result
	IF eTestResult = E_CommandResult.Ok THEN
		AssertEquals_UDINT(
			Expected := E_CommandState.Complete,
			Actual := iTestCommand.P_CommandStatus.StepState,
			Message := CONCAT(sTestScenario, ': STATE - Ok result should be in Complete state')
		);
	ELSE
		AssertEquals_UDINT(
			Expected := E_CommandState.Idle,
			Actual := iTestCommand.P_CommandStatus.StepState,
			Message := CONCAT(sTestScenario, ': STATE - Error results should return to Idle state')
		);
	END_IF

